LIN {X 0,Y 312.463,Z 248.062,A -85,B 0,C 180,E1 -15613.962,E2 -15613.962} C_VEL
LIN {X 0,Y 312.46,Z 248.062,A -85,B 0,C 180,E1 -15617.921,E2 -15617.921} C_VEL
LIN {X 0,Y 312.479,Z 248.055,A -85,B 0,C 180,E1 -15621.921,E2 -15621.921} C_VEL
LIN {X 0,Y 312.532,Z 248.051,A -85,B 0,C 180,E1 -15624.216,E2 -15624.216} C_VEL
LIN {X 0,Y 312.504,Z 248.056,A -85,B 0,C 180,E1 -15627.33,E2 -15627.33} C_VEL
LIN {X 0,Y 312.506,Z 248.055,A -85,B 0,C 180,E1 -15631.289,E2 -15631.289} C_VEL
LIN {X 0,Y 312.546,Z 248.054,A -85,B 0,C 180,E1 -15634.704,E2 -15634.704} C_VEL
LIN {X 0,Y 312.532,Z 248.054,A -85,B 0,C 180,E1 -15638.908,E2 -15638.908} C_VEL
LIN {X 0,Y 312.587,Z 248.036,A -85,B 0,C 180,E1 -15641.649,E2 -15641.649} C_VEL
LIN {X 0,Y 312.682,Z 248.028,A -85,B 0,C 180,E1 -15645.682,E2 -15645.682} C_VEL
LIN {X 0,Y 312.68,Z 248.034,A -85,B 0,C 180,E1 -15649.637,E2 -15649.637} C_VEL
LIN {X 0,Y 312.811,Z 248.012,A -85,B 0,C 180,E1 -15652.249,E2 -15652.249} C_VEL
LIN {X 0,Y 312.682,Z 248.035,A -85,B 0,C 180,E1 -15654.838,E2 -15654.838} C_VEL
LIN {X 0,Y 312.97,Z 247.999,A -85,B 0,C 180,E1 -15658.709,E2 -15658.709} C_VEL
LIN {X 0,Y 312.953,Z 247.992,A -85,B 0,C 180,E1 -15661.282,E2 -15661.282} C_VEL
LIN {X 0,Y 312.826,Z 248.014,A -85,B 0,C 180,E1 -15666.445,E2 -15666.445} C_VEL
LIN {X 0,Y 312.738,Z 248.025,A -85,B 0,C 180,E1 -15669.046,E2 -15669.046} C_VEL
LIN {X 0,Y 312.618,Z 248.04,A -85,B 0,C 180,E1 -15672.987,E2 -15672.987} C_VEL
LIN {X 0,Y 312.61,Z 248.048,A -85,B 0,C 180,E1 -15675.646,E2 -15675.646} C_VEL
LIN {X 0,Y 312.547,Z 248.051,A -85,B 0,C 180,E1 -15679.707,E2 -15679.707} C_VEL
LIN {X 0,Y 312.504,Z 248.054,A -85,B 0,C 180,E1 -15682.775,E2 -15682.775} C_VEL
LIN {X 0,Y 312.511,Z 248.055,A -85,B 0,C 180,E1 -15685.904,E2 -15685.904} C_VEL
LIN {X 0,Y 312.474,Z 248.056,A -85,B 0,C 180,E1 -15689.651,E2 -15689.651} C_VEL
LIN {X 0,Y 312.496,Z 248.061,A -85,B 0,C 180,E1 -15693.685,E2 -15693.685} C_VEL
LIN {X 0,Y 312.517,Z 248.195,A -85,B 0,C 180,E1 -15696.503,E2 -15696.503} C_VEL
LIN {X 0,Y 314.901,Z 258.143,A -85,B 0,C 180,E1 -15699.907,E2 -15699.907} C_VEL
LIN {X 0,Y 315.377,Z 260.256,A -85,B 0,C 180,E1 -15700.485,E2 -15700.485} C_VEL
LIN {X 0,Y 322.558,Z 277.103,A -85,B 0,C 180,E1 -15701.66,E2 -15701.66} C_VEL
LIN {X 0,Y 325.828,Z 294.759,A -85,B 0,C 180,E1 -15702.408,E2 -15702.408} C_VEL
LIN {X 0,Y 323.737,Z 367.932,A -85,B 0,C 180,E1 -15704.094,E2 -15704.094} C_VEL
LIN {X 0,Y 322.887,Z 381.785,A -85,B 0,C 180,E1 -15704.674,E2 -15704.674} C_VEL
LIN {X 0,Y 321.877,Z 394.277,A -85,B 0,C 180,E1 -15705.46,E2 -15705.46} C_VEL
LIN {X 0,Y 320.612,Z 405.801,A -85,B 0,C 180,E1 -15706.439,E2 -15706.439} C_VEL
LIN {X 0,Y 319.215,Z 416.53,A -85,B 0,C 180,E1 -15707.605,E2 -15707.605} C_VEL
LIN {X 0,Y 317.574,Z 427.06,A -85,B 0,C 180,E1 -15709.033,E2 -15709.033} C_VEL
LIN {X 0,Y 316.045,Z 436.49,A -85,B 0,C 180,E1 -15710.635,E2 -15710.635} C_VEL
LIN {X 0,Y 314.588,Z 445.259,A -85,B 0,C 180,E1 -15712.501,E2 -15712.501} C_VEL
LIN {X 0,Y 313.392,Z 452.216,A -85,B 0,C 180,E1 -15714.335,E2 -15714.335} C_VEL
LIN {X 0,Y 312.34,Z 458.327,A -85,B 0,C 180,E1 -15716.35,E2 -15716.35} C_VEL
LIN {X 0,Y 311.51,Z 463.814,A -85,B 0,C 180,E1 -15718.743,E2 -15718.743} C_VEL
LIN {X 0,Y 311.136,Z 466.376,A -85,B 0,C 180,E1 -15720.204,E2 -15720.204} C_VEL
LIN {X 0,Y 310.784,Z 468.579,A -85,B 0,C 180,E1 -15721.864,E2 -15721.864} C_VEL
LIN {X 0,Y 310.578,Z 469.776,A -85,B 0,C 180,E1 -15723.092,E2 -15723.092} C_VEL
LIN {X 0,Y 310.4,Z 470.87,A -85,B 0,C 180,E1 -15724.899,E2 -15724.899} C_VEL
LIN {X 0,Y 310.274,Z 471.125,A -85,B 0,C 180,E1 -15727.354,E2 -15727.354} C_VEL
LIN {X 0,Y 310.36,Z 470.641,A -85,B 0,C 180,E1 -15728.759,E2 -15728.759} C_VEL
LIN {X 0,Y 310.458,Z 469.66,A -85,B 0,C 180,E1 -15730.151,E2 -15730.151} C_VEL
LIN {X 0,Y 310.677,Z 467.93,A -85,B 0,C 180,E1 -15731.804,E2 -15731.804} C_VEL
LIN {X 0,Y 310.973,Z 465.238,A -85,B 0,C 180,E1 -15733.592,E2 -15733.592} C_VEL
LIN {X 0,Y 311.569,Z 460.486,A -85,B 0,C 180,E1 -15735.89,E2 -15735.89} C_VEL
LIN {X 0,Y 312.285,Z 454.707,A -85,B 0,C 180,E1 -15737.986,E2 -15737.986} C_VEL
LIN {X 0,Y 313.308,Z 447.063,A -85,B 0,C 180,E1 -15740.153,E2 -15740.153} C_VEL
LIN {X 0,Y 314.507,Z 438.905,A -85,B 0,C 180,E1 -15741.973,E2 -15741.973} C_VEL
LIN {X 0,Y 315.903,Z 428.823,A -85,B 0,C 180,E1 -15743.775,E2 -15743.775} C_VEL
LIN {X 0,Y 317.304,Z 418.3,A -85,B 0,C 180,E1 -15745.273,E2 -15745.273} C_VEL
LIN {X 0,Y 318.603,Z 407.173,A -85,B 0,C 180,E1 -15746.523,E2 -15746.523} C_VEL
LIN {X 0,Y 319.848,Z 394.355,A -85,B 0,C 180,E1 -15747.64,E2 -15747.64} C_VEL
LIN {X 0,Y 320.764,Z 381.876,A -85,B 0,C 180,E1 -15748.432,E2 -15748.432} C_VEL
LIN {X 0,Y 321.492,Z 369.025,A -85,B 0,C 180,E1 -15748.983,E2 -15748.983} C_VEL
LIN {X 0,Y 322.286,Z 339.702,A -85,B 0,C 180,E1 -15749.689,E2 -15749.689} C_VEL
LIN {X 0,Y 323.282,Z 292.285,A -85,B 0,C 180,E1 -15750.766,E2 -15750.766} C_VEL
LIN {X 0,Y 319.172,Z 270.918,A -85,B 0,C 180,E1 -15751.59,E2 -15751.59} C_VEL
LIN {X 0,Y 315.333,Z 260.355,A -85,B 0,C 180,E1 -15752.181,E2 -15752.181} C_VEL
LIN {X 0,Y 314.589,Z 256.888,A -85,B 0,C 180,E1 -15753.203,E2 -15753.203} C_VEL
LIN {X 0,Y 312.881,Z 248.091,A -85,B 0,C 180,E1 -15756.207,E2 -15756.207} C_VEL
LIN {X 0,Y 312.734,Z 248.024,A -85,B 0,C 180,E1 -15759.052,E2 -15759.052} C_VEL
LIN {X 0,Y 312.603,Z 248.034,A -85,B 0,C 180,E1 -15762.993,E2 -15762.993} C_VEL
LIN {X 0,Y 312.607,Z 248.043,A -85,B 0,C 180,E1 -15765.652,E2 -15765.652} C_VEL
LIN {X 0,Y 312.578,Z 248.046,A -85,B 0,C 180,E1 -15769.227,E2 -15769.227} C_VEL
LIN {X 0,Y 312.492,Z 248.057,A -85,B 0,C 180,E1 -15772.781,E2 -15772.781} C_VEL
LIN {X 0,Y 312.502,Z 248.057,A -85,B 0,C 180,E1 -15775.911,E2 -15775.911} C_VEL
LIN {X 0,Y 312.445,Z 248.051,A -85,B 0,C 180,E1 -15779.661,E2 -15779.661} C_VEL
LIN {X 0,Y 312.494,Z 248.056,A -85,B 0,C 180,E1 -15783.693,E2 -15783.693} C_VEL
LIN {X 0,Y 312.485,Z 248.057,A -85,B 0,C 180,E1 -15787.392,E2 -15787.392} C_VEL
LIN {X 0,Y 312.402,Z 248.056,A -85,B 0,C 180,E1 -15791.155,E2 -15791.155} C_VEL
LIN {X 0,Y 311.733,Z 248.136,A -85,B 0,C 180,E1 -15792.231,E2 -15792.231} C_VEL
LIN {X 0,Y 308.889,Z 248.495,A -85,B 0,C 180,E1 -15793.983,E2 -15793.983} C_VEL
LIN {X 0,Y 306.488,Z 248.805,A -85,B 0,C 180,E1 -15795.404,E2 -15795.404} C_VEL
LIN {X 0,Y 305.47,Z 248.934,A -85,B 0,C 180,E1 -15796.504,E2 -15796.504} C_VEL
LIN {X 0,Y 305.394,Z 248.94,A -85,B 0,C 180,E1 -15796.877,E2 -15796.877} C_VEL
LIN {X 0,Y 305.392,Z 248.928,A -85,B 0,C 180,E1 -15799.889,E2 -15799.889} C_VEL
LIN {X 0,Y 305.446,Z 248.929,A -85,B 0,C 180,E1 -15803.642,E2 -15803.642} C_VEL
LIN {X 0,Y 305.451,Z 248.935,A -85,B 0,C 180,E1 -15806.488,E2 -15806.488} C_VEL
LIN {X 0,Y 305.404,Z 248.92,A -85,B 0,C 180,E1 -15809.591,E2 -15809.591} C_VEL
LIN {X 0,Y 305.43,Z 248.914,A -85,B 0,C 180,E1 -15812.606,E2 -15812.606} C_VEL
LIN {X 0,Y 305.446,Z 248.936,A -85,B 0,C 180,E1 -15815.539,E2 -15815.539} C_VEL
LIN {X 0,Y 305.489,Z 248.916,A -85,B 0,C 180,E1 -15819.818,E2 -15819.818} C_VEL
LIN {X 0,Y 305.536,Z 248.886,A -85,B 0,C 180,E1 -15822.606,E2 -15822.606} C_VEL
LIN {X 0,Y 305.622,Z 248.9,A -85,B 0,C 180,E1 -15825.353,E2 -15825.353} C_VEL
LIN {X 0,Y 305.621,Z 248.914,A -85,B 0,C 180,E1 -15829.404,E2 -15829.404} C_VEL
LIN {X 0,Y 305.745,Z 248.876,A -85,B 0,C 180,E1 -15832.077,E2 -15832.077} C_VEL
LIN {X 0,Y 305.657,Z 248.877,A -85,B 0,C 180,E1 -15834.728,E2 -15834.728} C_VEL
LIN {X 0,Y 305.937,Z 248.873,A -85,B 0,C 180,E1 -15838.688,E2 -15838.688} C_VEL
LIN {X 0,Y 305.947,Z 248.868,A -85,B 0,C 180,E1 -15841.321,E2 -15841.321} C_VEL
LIN {X 0,Y 305.809,Z 248.866,A -85,B 0,C 180,E1 -15846.603,E2 -15846.603} C_VEL
LIN {X 0,Y 305.701,Z 248.902,A -85,B 0,C 180,E1 -15849.265,E2 -15849.265} C_VEL
LIN {X 0,Y 305.593,Z 248.905,A -85,B 0,C 180,E1 -15853.3,E2 -15853.3} C_VEL
LIN {X 0,Y 305.56,Z 248.898,A -85,B 0,C 180,E1 -15856.026,E2 -15856.026} C_VEL
LIN {X 0,Y 305.552,Z 248.923,A -85,B 0,C 180,E1 -15859.43,E2 -15859.43} C_VEL
LIN {X 0,Y 305.497,Z 248.911,A -85,B 0,C 180,E1 -15863.042,E2 -15863.042} C_VEL
LIN {X 0,Y 305.481,Z 248.926,A -85,B 0,C 180,E1 -15866.2,E2 -15866.2} C_VEL
LIN {X 0,Y 305.46,Z 248.933,A -85,B 0,C 180,E1 -15869.036,E2 -15869.036} C_VEL
LIN {X 0,Y 305.448,Z 248.924,A -85,B 0,C 180,E1 -15871.956,E2 -15871.956} C_VEL
LIN {X 0,Y 305.474,Z 248.936,A -85,B 0,C 180,E1 -15875.116,E2 -15875.116} C_VEL
LIN {X 0,Y 305.446,Z 248.93,A -85,B 0,C 180,E1 -15878.527,E2 -15878.527} C_VEL
LIN {X 0,Y 305.448,Z 248.925,A -85,B 0,C 180,E1 -15882.583,E2 -15882.583} C_VEL
LIN {X 0,Y 305.434,Z 248.933,A -85,B 0,C 180,E1 -15886.345,E2 -15886.345} C_VEL
LIN {X 0,Y 305.424,Z 248.938,A -85,B 0,C 180,E1 -15889.886,E2 -15889.886} C_VEL
LIN {X 0,Y 305.476,Z 248.933,A -85,B 0,C 180,E1 -15893.638,E2 -15893.638} C_VEL
LIN {X 0,Y 305.479,Z 248.924,A -85,B 0,C 180,E1 -15896.484,E2 -15896.484} C_VEL
LIN {X 0,Y 305.471,Z 248.993,A -85,B 0,C 180,E1 -15898.211,E2 -15898.211} C_VEL
LIN {X 0,Y 307.479,Z 258.119,A -85,B 0,C 180,E1 -15901.314,E2 -15901.314} C_VEL
LIN {X 0,Y 309.395,Z 267.921,A -85,B 0,C 180,E1 -15904.363,E2 -15904.363} C_VEL
LIN {X 0,Y 310.742,Z 272.023,A -85,B 0,C 180,E1 -15904.643,E2 -15904.643} C_VEL
LIN {X 0,Y 315.958,Z 302.066,A -85,B 0,C 180,E1 -15905.787,E2 -15905.787} C_VEL
LIN {X 0,Y 316.558,Z 306.759,A -85,B 0,C 180,E1 -15905.946,E2 -15905.946} C_VEL
LIN {X 0,Y 314.819,Z 376.369,A -85,B 0,C 180,E1 -15907.581,E2 -15907.581} C_VEL
LIN {X 0,Y 314.013,Z 389.829,A -85,B 0,C 180,E1 -15908.155,E2 -15908.155} C_VEL
LIN {X 0,Y 312.93,Z 402.282,A -85,B 0,C 180,E1 -15908.939,E2 -15908.939} C_VEL
LIN {X 0,Y 311.745,Z 413.411,A -85,B 0,C 180,E1 -15909.891,E2 -15909.891} C_VEL
LIN {X 0,Y 310.33,Z 425.013,A -85,B 0,C 180,E1 -15911.172,E2 -15911.172} C_VEL
LIN {X 0,Y 308.952,Z 435.464,A -85,B 0,C 180,E1 -15912.628,E2 -15912.628} C_VEL
LIN {X 0,Y 307.797,Z 444.002,A -85,B 0,C 180,E1 -15914.097,E2 -15914.097} C_VEL
LIN {X 0,Y 306.403,Z 453.236,A -85,B 0,C 180,E1 -15916.063,E2 -15916.063} C_VEL
LIN {X 0,Y 305.282,Z 460.656,A -85,B 0,C 180,E1 -15918.041,E2 -15918.041} C_VEL
LIN {X 0,Y 304.54,Z 466.605,A -85,B 0,C 180,E1 -15920.032,E2 -15920.032} C_VEL
LIN {X 0,Y 304.022,Z 471.29,A -85,B 0,C 180,E1 -15922.026,E2 -15922.026} C_VEL
LIN {X 0,Y 303.673,Z 475.387,A -85,B 0,C 180,E1 -15924.387,E2 -15924.387} C_VEL
LIN {X 0,Y 303.596,Z 477.39,A -85,B 0,C 180,E1 -15926.017,E2 -15926.017} C_VEL
LIN {X 0,Y 303.586,Z 478.574,A -85,B 0,C 180,E1 -15927.345,E2 -15927.345} C_VEL
LIN {X 0,Y 303.534,Z 479.309,A -85,B 0,C 180,E1 -15928.672,E2 -15928.672} C_VEL
LIN {X 0,Y 303.541,Z 479.653,A -85,B 0,C 180,E1 -15929.999,E2 -15929.999} C_VEL
LIN {X 0,Y 303.534,Z 479.61,A -85,B 0,C 180,E1 -15931.326,E2 -15931.326} C_VEL
LIN {X 0,Y 303.588,Z 479.175,A -85,B 0,C 180,E1 -15932.653,E2 -15932.653} C_VEL
LIN {X 0,Y 303.606,Z 478.302,A -85,B 0,C 180,E1 -15933.981,E2 -15933.981} C_VEL
LIN {X 0,Y 303.849,Z 475.356,A -85,B 0,C 180,E1 -15936.64,E2 -15936.64} C_VEL
LIN {X 0,Y 304.242,Z 471.997,A -85,B 0,C 180,E1 -15938.634,E2 -15938.634} C_VEL
LIN {X 0,Y 304.898,Z 467.57,A -85,B 0,C 180,E1 -15940.625,E2 -15940.625} C_VEL
LIN {X 0,Y 305.793,Z 461.955,A -85,B 0,C 180,E1 -15942.61,E2 -15942.61} C_VEL
LIN {X 0,Y 307.091,Z 454.946,A -85,B 0,C 180,E1 -15944.579,E2 -15944.579} C_VEL
LIN {X 0,Y 308.657,Z 446.316,A -85,B 0,C 180,E1 -15946.507,E2 -15946.507} C_VEL
LIN {X 0,Y 310.224,Z 436.252,A -85,B 0,C 180,E1 -15948.319,E2 -15948.319} C_VEL
LIN {X 0,Y 311.905,Z 426.151,A -85,B 0,C 180,E1 -15949.753,E2 -15949.753} C_VEL
LIN {X 0,Y 313.56,Z 414.959,A -85,B 0,C 180,E1 -15951.014,E2 -15951.014} C_VEL
LIN {X 0,Y 315.056,Z 402.422,A -85,B 0,C 180,E1 -15952.112,E2 -15952.112} C_VEL
LIN {X 0,Y 316.337,Z 389.519,A -85,B 0,C 180,E1 -15952.921,E2 -15952.921} C_VEL
LIN {X 0,Y 317.264,Z 375.829,A -85,B 0,C 180,E1 -15953.498,E2 -15953.498} C_VEL
LIN {X 0,Y 319.018,Z 315.952,A -85,B 0,C 180,E1 -15954.913,E2 -15954.913} C_VEL
LIN {X 0,Y 319.112,Z 306.429,A -85,B 0,C 180,E1 -15955.15,E2 -15955.15} C_VEL
LIN {X 0,Y 315.545,Z 285.854,A -85,B 0,C 180,E1 -15956.032,E2 -15956.032} C_VEL
LIN {X 0,Y 313.593,Z 277.044,A -85,B 0,C 180,E1 -15956.463,E2 -15956.463} C_VEL
LIN {X 0,Y 309.713,Z 267.394,A -85,B 0,C 180,E1 -15957.172,E2 -15957.172} C_VEL
LIN {X 0,Y 307.708,Z 258.136,A -85,B 0,C 180,E1 -15960.162,E2 -15960.162} C_VEL
LIN {X 0,Y 305.518,Z 248.992,A -85,B 0,C 180,E1 -15963.459,E2 -15963.459} C_VEL
LIN {X 0,Y 305.461,Z 248.927,A -85,B 0,C 180,E1 -15966.74,E2 -15966.74} C_VEL
LIN {X 0,Y 305.416,Z 248.93,A -85,B 0,C 180,E1 -15970.587,E2 -15970.587} C_VEL
LIN {X 0,Y 305.427,Z 248.936,A -85,B 0,C 180,E1 -15973.653,E2 -15973.653} C_VEL
LIN {X 0,Y 305.44,Z 248.938,A -85,B 0,C 180,E1 -15977.415,E2 -15977.415} C_VEL
LIN {X 0,Y 305.445,Z 248.93,A -85,B 0,C 180,E1 -15981.589,E2 -15981.589} C_VEL
LIN {X 0,Y 305.464,Z 248.929,A -85,B 0,C 180,E1 -15984.883,E2 -15984.883} C_VEL
LIN {X 0,Y 305.444,Z 248.931,A -85,B 0,C 180,E1 -15988.355,E2 -15988.355} C_VEL
LIN {X 0,Y 305.475,Z 248.932,A -85,B 0,C 180,E1 -15991.105,E2 -15991.105} C_VEL
LIN {X 0,Y 305.498,Z 248.927,A -85,B 0,C 180,E1 -15994.077,E2 -15994.077} C_VEL
LIN {X 0,Y 305.474,Z 248.924,A -85,B 0,C 180,E1 -15996.972,E2 -15996.972} C_VEL
LIN {X 0,Y 305.547,Z 248.914,A -85,B 0,C 180,E1 -16001.211,E2 -16001.211} C_VEL
LIN {X 0,Y 305.623,Z 248.909,A -85,B 0,C 180,E1 -16005.344,E2 -16005.344} C_VEL
LIN {X 0,Y 305.619,Z 248.916,A -85,B 0,C 180,E1 -16009.395,E2 -16009.395} C_VEL
LIN {X 0,Y 305.757,Z 248.889,A -85,B 0,C 180,E1 -16012.069,E2 -16012.069} C_VEL
LIN {X 0,Y 305.653,Z 248.911,A -85,B 0,C 180,E1 -16014.719,E2 -16014.719} C_VEL
LIN {X 0,Y 305.936,Z 248.875,A -85,B 0,C 180,E1 -16018.679,E2 -16018.679} C_VEL
LIN {X 0,Y 305.921,Z 248.868,A -85,B 0,C 180,E1 -16021.312,E2 -16021.312} C_VEL
LIN {X 0,Y 305.771,Z 248.894,A -85,B 0,C 180,E1 -16026.594,E2 -16026.594} C_VEL
LIN {X 0,Y 305.681,Z 248.902,A -85,B 0,C 180,E1 -16029.257,E2 -16029.257} C_VEL
LIN {X 0,Y 305.57,Z 248.917,A -85,B 0,C 180,E1 -16033.292,E2 -16033.292} C_VEL
LIN {X 0,Y 305.539,Z 248.925,A -85,B 0,C 180,E1 -16036.018,E2 -16036.018} C_VEL
LIN {X 0,Y 305.53,Z 248.927,A -85,B 0,C 180,E1 -16039.424,E2 -16039.424} C_VEL
LIN {X 0,Y 305.468,Z 248.93,A -85,B 0,C 180,E1 -16043.035,E2 -16043.035} C_VEL
LIN {X 0,Y 305.451,Z 248.937,A -85,B 0,C 180,E1 -16046.193,E2 -16046.193} C_VEL
LIN {X 0,Y 305.427,Z 248.928,A -85,B 0,C 180,E1 -16049.03,E2 -16049.03} C_VEL
LIN {X 0,Y 305.414,Z 248.933,A -85,B 0,C 180,E1 -16051.949,E2 -16051.949} C_VEL
LIN {X 0,Y 305.515,Z 249.124,A -85,B 0,C 180,E1 -16055.913,E2 -16055.913} C_VEL
LIN {X 0,Y 307.844,Z 258.921,A -85,B 0,C 180,E1 -16059.366,E2 -16059.366} C_VEL
LIN {X 0,Y 308.209,Z 260.311,A -85,B 0,C 180,E1 -16059.734,E2 -16059.734} C_VEL
LIN {X 0,Y 315.471,Z 276.995,A -85,B 0,C 180,E1 -16060.969,E2 -16060.969} C_VEL
LIN {X 0,Y 316.962,Z 281.432,A -85,B 0,C 180,E1 -16061.233,E2 -16061.233} C_VEL
LIN {X 0,Y 319.506,Z 295.751,A -85,B 0,C 180,E1 -16061.852,E2 -16061.852} C_VEL
LIN {X 0,Y 317.415,Z 367.051,A -85,B 0,C 180,E1 -16063.522,E2 -16063.522} C_VEL
LIN {X 0,Y 316.594,Z 380.179,A -85,B 0,C 180,E1 -16064.056,E2 -16064.056} C_VEL
LIN {X 0,Y 315.55,Z 392.768,A -85,B 0,C 180,E1 -16064.828,E2 -16064.828} C_VEL
LIN {X 0,Y 314.231,Z 404.522,A -85,B 0,C 180,E1 -16065.801,E2 -16065.801} C_VEL
LIN {X 0,Y 312.784,Z 415.314,A -85,B 0,C 180,E1 -16066.963,E2 -16066.963} C_VEL
LIN {X 0,Y 311.074,Z 426.08,A -85,B 0,C 180,E1 -16068.419,E2 -16068.419} C_VEL
LIN {X 0,Y 309.412,Z 435.917,A -85,B 0,C 180,E1 -16070.085,E2 -16070.085} C_VEL
LIN {X 0,Y 307.858,Z 444.664,A -85,B 0,C 180,E1 -16071.95,E2 -16071.95} C_VEL
LIN {X 0,Y 306.598,Z 451.752,A -85,B 0,C 180,E1 -16073.827,E2 -16073.827} C_VEL
LIN {X 0,Y 305.474,Z 458.032,A -85,B 0,C 180,E1 -16075.908,E2 -16075.908} C_VEL
LIN {X 0,Y 304.649,Z 462.849,A -85,B 0,C 180,E1 -16077.956,E2 -16077.956} C_VEL
LIN {X 0,Y 304.038,Z 466.792,A -85,B 0,C 180,E1 -16080.201,E2 -16080.201} C_VEL
LIN {X 0,Y 303.579,Z 469.427,A -85,B 0,C 180,E1 -16082.42,E2 -16082.42} C_VEL
LIN {X 0,Y 303.329,Z 470.904,A -85,B 0,C 180,E1 -16084.622,E2 -16084.622} C_VEL
LIN {X 0,Y 303.181,Z 471.291,A -85,B 0,C 180,E1 -16086.793,E2 -16086.793} C_VEL
LIN {X 0,Y 303.252,Z 470.953,A -85,B 0,C 180,E1 -16088.236,E2 -16088.236} C_VEL
LIN {X 0,Y 303.305,Z 470.184,A -85,B 0,C 180,E1 -16089.663,E2 -16089.663} C_VEL
LIN {X 0,Y 303.564,Z 468.295,A -85,B 0,C 180,E1 -16091.641,E2 -16091.641} C_VEL
LIN {X 0,Y 303.933,Z 465.019,A -85,B 0,C 180,E1 -16093.891,E2 -16093.891} C_VEL
LIN {X 0,Y 304.581,Z 460.129,A -85,B 0,C 180,E1 -16096.237,E2 -16096.237} C_VEL
LIN {X 0,Y 305.339,Z 454.229,A -85,B 0,C 180,E1 -16098.382,E2 -16098.382} C_VEL
LIN {X 0,Y 306.383,Z 446.861,A -85,B 0,C 180,E1 -16100.487,E2 -16100.487} C_VEL
LIN {X 0,Y 307.698,Z 438.079,A -85,B 0,C 180,E1 -16102.455,E2 -16102.455} C_VEL
LIN {X 0,Y 309.063,Z 428.803,A -85,B 0,C 180,E1 -16104.128,E2 -16104.128} C_VEL
LIN {X 0,Y 310.411,Z 418.956,A -85,B 0,C 180,E1 -16105.566,E2 -16105.566} C_VEL
LIN {X 0,Y 311.855,Z 407.074,A -85,B 0,C 180,E1 -16106.933,E2 -16106.933} C_VEL
LIN {X 0,Y 313.045,Z 395.22,A -85,B 0,C 180,E1 -16107.991,E2 -16107.991} C_VEL
LIN {X 0,Y 313.998,Z 383.123,A -85,B 0,C 180,E1 -16108.799,E2 -16108.799} C_VEL
LIN {X 0,Y 314.79,Z 369.706,A -85,B 0,C 180,E1 -16109.401,E2 -16109.401} C_VEL
LIN {X 0,Y 315.518,Z 347.471,A -85,B 0,C 180,E1 -16109.961,E2 -16109.961} C_VEL
LIN {X 0,Y 316.669,Z 293.156,A -85,B 0,C 180,E1 -16111.224,E2 -16111.224} C_VEL
LIN {X 0,Y 312.829,Z 273.23,A -85,B 0,C 180,E1 -16112.013,E2 -16112.013} C_VEL
LIN {X 0,Y 308.164,Z 260.505,A -85,B 0,C 180,E1 -16112.738,E2 -16112.738} C_VEL
LIN {X 0,Y 307.685,Z 258.533,A -85,B 0,C 180,E1 -16113.275,E2 -16113.275} C_VEL
LIN {X 0,Y 305.844,Z 248.989,A -85,B 0,C 180,E1 -16116.599,E2 -16116.599} C_VEL
LIN {X 0,Y 305.671,Z 248.903,A -85,B 0,C 180,E1 -16119.263,E2 -16119.263} C_VEL
LIN {X 0,Y 305.557,Z 248.913,A -85,B 0,C 180,E1 -16123.298,E2 -16123.298} C_VEL
LIN {X 0,Y 305.562,Z 248.918,A -85,B 0,C 180,E1 -16126.023,E2 -16126.023} C_VEL
LIN {X 0,Y 305.529,Z 248.922,A -85,B 0,C 180,E1 -16129.438,E2 -16129.438} C_VEL
LIN {X 0,Y 305.457,Z 248.933,A -85,B 0,C 180,E1 -16133.043,E2 -16133.043} C_VEL
LIN {X 0,Y 305.442,Z 248.939,A -85,B 0,C 180,E1 -16136.201,E2 -16136.201} C_VEL
LIN {X 0,Y 305.408,Z 248.927,A -85,B 0,C 180,E1 -16139.033,E2 -16139.033} C_VEL
LIN {X 0,Y 305.409,Z 248.942,A -85,B 0,C 180,E1 -16141.957,E2 -16141.957} C_VEL
LIN {X 0,Y 305.435,Z 248.92,A -85,B 0,C 180,E1 -16145.118,E2 -16145.118} C_VEL
LIN {X 0,Y 305.41,Z 248.944,A -85,B 0,C 180,E1 -16148.529,E2 -16148.529} C_VEL
LIN {X 0,Y 305.412,Z 248.921,A -85,B 0,C 180,E1 -16152.586,E2 -16152.586} C_VEL
LIN {X 0,Y 305.394,Z 248.94,A -85,B 0,C 180,E1 -16156.877,E2 -16156.877} C_VEL
LIN {X 0,Y 304.737,Z 249.024,A -85,B 0,C 180,E1 -16157.978,E2 -16157.978} C_VEL
LIN {X 0,Y 301.874,Z 249.366,A -85,B 0,C 180,E1 -16159.771,E2 -16159.771} C_VEL
LIN {X 0,Y 299.457,Z 249.659,A -85,B 0,C 180,E1 -16161.226,E2 -16161.226} C_VEL
LIN {X 0,Y 298.447,Z 249.785,A -85,B 0,C 180,E1 -16162.353,E2 -16162.353} C_VEL
LIN {X 0,Y 298.38,Z 249.796,A -85,B 0,C 180,E1 -16162.735,E2 -16162.735} C_VEL
LIN {X 0,Y 298.393,Z 249.814,A -85,B 0,C 180,E1 -16165.586,E2 -16165.586} C_VEL
LIN {X 0,Y 298.359,Z 249.807,A -85,B 0,C 180,E1 -16168.794,E2 -16168.794} C_VEL
LIN {X 0,Y 298.384,Z 249.785,A -85,B 0,C 180,E1 -16171.902,E2 -16171.902} C_VEL
LIN {X 0,Y 298.412,Z 249.806,A -85,B 0,C 180,E1 -16174.923,E2 -16174.923} C_VEL
LIN {X 0,Y 298.419,Z 249.801,A -85,B 0,C 180,E1 -16179.319,E2 -16179.319} C_VEL
LIN {X 0,Y 298.472,Z 249.766,A -85,B 0,C 180,E1 -16182.181,E2 -16182.181} C_VEL
LIN {X 0,Y 298.583,Z 249.775,A -85,B 0,C 180,E1 -16184.999,E2 -16184.999} C_VEL
LIN {X 0,Y 298.58,Z 249.79,A -85,B 0,C 180,E1 -16189.151,E2 -16189.151} C_VEL
LIN {X 0,Y 298.696,Z 249.755,A -85,B 0,C 180,E1 -16191.889,E2 -16191.889} C_VEL
LIN {X 0,Y 298.627,Z 249.751,A -85,B 0,C 180,E1 -16194.603,E2 -16194.603} C_VEL
LIN {X 0,Y 298.905,Z 249.749,A -85,B 0,C 180,E1 -16198.657,E2 -16198.657} C_VEL
LIN {X 0,Y 298.914,Z 249.745,A -85,B 0,C 180,E1 -16201.352,E2 -16201.352} C_VEL
LIN {X 0,Y 298.758,Z 249.746,A -85,B 0,C 180,E1 -16206.759,E2 -16206.759} C_VEL
LIN {X 0,Y 298.632,Z 249.783,A -85,B 0,C 180,E1 -16209.486,E2 -16209.486} C_VEL
LIN {X 0,Y 298.552,Z 249.781,A -85,B 0,C 180,E1 -16213.62,E2 -16213.62} C_VEL
LIN {X 0,Y 298.495,Z 249.78,A -85,B 0,C 180,E1 -16216.416,E2 -16216.416} C_VEL
LIN {X 0,Y 298.493,Z 249.802,A -85,B 0,C 180,E1 -16219.642,E2 -16219.642} C_VEL
LIN {X 0,Y 298.431,Z 249.786,A -85,B 0,C 180,E1 -16223.604,E2 -16223.604} C_VEL
LIN {X 0,Y 298.419,Z 249.807,A -85,B 0,C 180,E1 -16226.585,E2 -16226.585} C_VEL
LIN {X 0,Y 298.405,Z 249.806,A -85,B 0,C 180,E1 -16229.647,E2 -16229.647} C_VEL
LIN {X 0,Y 298.405,Z 249.805,A -85,B 0,C 180,E1 -16232.803,E2 -16232.803} C_VEL
LIN {X 0,Y 298.439,Z 249.801,A -85,B 0,C 180,E1 -16236.804,E2 -16236.804} C_VEL
LIN {X 0,Y 298.387,Z 249.816,A -85,B 0,C 180,E1 -16239.494,E2 -16239.494} C_VEL
LIN {X 0,Y 298.383,Z 249.807,A -85,B 0,C 180,E1 -16243.099,E2 -16243.099} C_VEL
LIN {X 0,Y 298.384,Z 249.812,A -85,B 0,C 180,E1 -16246.916,E2 -16246.916} C_VEL
LIN {X 0,Y 298.399,Z 249.816,A -85,B 0,C 180,E1 -16251.012,E2 -16251.012} C_VEL
LIN {X 0,Y 298.418,Z 249.812,A -85,B 0,C 180,E1 -16253.929,E2 -16253.929} C_VEL
LIN {X 0,Y 298.417,Z 249.875,A -85,B 0,C 180,E1 -16257.768,E2 -16257.768} C_VEL
LIN {X 0,Y 300.444,Z 259.031,A -85,B 0,C 180,E1 -16260.961,E2 -16260.961} C_VEL
LIN {X 0,Y 302.159,Z 267.831,A -85,B 0,C 180,E1 -16263.772,E2 -16263.772} C_VEL
LIN {X 0,Y 303.904,Z 272.76,A -85,B 0,C 180,E1 -16264.112,E2 -16264.112} C_VEL
LIN {X 0,Y 305.261,Z 278.652,A -85,B 0,C 180,E1 -16264.375,E2 -16264.375} C_VEL
LIN {X 0,Y 309.848,Z 306.247,A -85,B 0,C 180,E1 -16265.437,E2 -16265.437} C_VEL
LIN {X 0,Y 308.263,Z 373.719,A -85,B 0,C 180,E1 -16267.048,E2 -16267.048} C_VEL
LIN {X 0,Y 307.527,Z 387.205,A -85,B 0,C 180,E1 -16267.581,E2 -16267.581} C_VEL
LIN {X 0,Y 306.39,Z 400.316,A -85,B 0,C 180,E1 -16268.379,E2 -16268.379} C_VEL
LIN {X 0,Y 305.051,Z 412.78,A -85,B 0,C 180,E1 -16269.43,E2 -16269.43} C_VEL
LIN {X 0,Y 303.574,Z 424.482,A -85,B 0,C 180,E1 -16270.736,E2 -16270.736} C_VEL
LIN {X 0,Y 302.152,Z 435.01,A -85,B 0,C 180,E1 -16272.224,E2 -16272.224} C_VEL
LIN {X 0,Y 300.937,Z 443.612,A -85,B 0,C 180,E1 -16273.724,E2 -16273.724} C_VEL
LIN {X 0,Y 299.729,Z 451.536,A -85,B 0,C 180,E1 -16275.399,E2 -16275.399} C_VEL
LIN {X 0,Y 298.499,Z 459.256,A -85,B 0,C 180,E1 -16277.42,E2 -16277.42} C_VEL
LIN {X 0,Y 297.514,Z 466.366,A -85,B 0,C 180,E1 -16279.794,E2 -16279.794} C_VEL
LIN {X 0,Y 296.973,Z 471.083,A -85,B 0,C 180,E1 -16281.836,E2 -16281.836} C_VEL
LIN {X 0,Y 296.749,Z 473.599,A -85,B 0,C 180,E1 -16283.198,E2 -16283.198} C_VEL
LIN {X 0,Y 296.565,Z 475.627,A -85,B 0,C 180,E1 -16284.56,E2 -16284.56} C_VEL
LIN {X 0,Y 296.499,Z 477.238,A -85,B 0,C 180,E1 -16285.921,E2 -16285.921} C_VEL
LIN {X 0,Y 296.491,Z 478.439,A -85,B 0,C 180,E1 -16287.282,E2 -16287.282} C_VEL
LIN {X 0,Y 296.456,Z 479.193,A -85,B 0,C 180,E1 -16288.64,E2 -16288.64} C_VEL
LIN {X 0,Y 296.459,Z 479.549,A -85,B 0,C 180,E1 -16289.999,E2 -16289.999} C_VEL
LIN {X 0,Y 296.456,Z 479.517,A -85,B 0,C 180,E1 -16291.357,E2 -16291.357} C_VEL
LIN {X 0,Y 296.493,Z 479.098,A -85,B 0,C 180,E1 -16292.716,E2 -16292.716} C_VEL
LIN {X 0,Y 296.51,Z 478.246,A -85,B 0,C 180,E1 -16294.076,E2 -16294.076} C_VEL
LIN {X 0,Y 296.599,Z 476.824,A -85,B 0,C 180,E1 -16295.588,E2 -16295.588} C_VEL
LIN {X 0,Y 297.032,Z 473.24,A -85,B 0,C 180,E1 -16298.16,E2 -16298.16} C_VEL
LIN {X 0,Y 297.624,Z 469.208,A -85,B 0,C 180,E1 -16300.2,E2 -16300.2} C_VEL
LIN {X 0,Y 298.696,Z 463.019,A -85,B 0,C 180,E1 -16302.569,E2 -16302.569} C_VEL
LIN {X 0,Y 299.992,Z 456.285,A -85,B 0,C 180,E1 -16304.585,E2 -16304.585} C_VEL
LIN {X 0,Y 301.604,Z 448.112,A -85,B 0,C 180,E1 -16306.545,E2 -16306.545} C_VEL
LIN {X 0,Y 303.046,Z 439.368,A -85,B 0,C 180,E1 -16308.243,E2 -16308.243} C_VEL
LIN {X 0,Y 304.658,Z 429.987,A -85,B 0,C 180,E1 -16309.716,E2 -16309.716} C_VEL
LIN {X 0,Y 306.556,Z 418.382,A -85,B 0,C 180,E1 -16311.165,E2 -16311.165} C_VEL
LIN {X 0,Y 308.049,Z 406.915,A -85,B 0,C 180,E1 -16312.288,E2 -16312.288} C_VEL
LIN {X 0,Y 309.526,Z 393.778,A -85,B 0,C 180,E1 -16313.234,E2 -16313.234} C_VEL
LIN {X 0,Y 310.641,Z 380.543,A -85,B 0,C 180,E1 -16313.897,E2 -16313.897} C_VEL
LIN {X 0,Y 311.336,Z 366.569,A -85,B 0,C 180,E1 -16314.308,E2 -16314.308} C_VEL
LIN {X 0,Y 312.832,Z 307.519,A -85,B 0,C 180,E1 -16315.725,E2 -16315.725} C_VEL
LIN {X 0,Y 309.162,Z 286.21,A -85,B 0,C 180,E1 -16316.668,E2 -16316.668} C_VEL
LIN {X 0,Y 307.655,Z 279.7,A -85,B 0,C 180,E1 -16317.007,E2 -16317.007} C_VEL
LIN {X 0,Y 302.505,Z 267.291,A -85,B 0,C 180,E1 -16317.957,E2 -16317.957} C_VEL
LIN {X 0,Y 300.527,Z 258.329,A -85,B 0,C 180,E1 -16320.961,E2 -16320.961} C_VEL
LIN {X 0,Y 298.467,Z 249.904,A -85,B 0,C 180,E1 -16324.103,E2 -16324.103} C_VEL
LIN {X 0,Y 298.405,Z 249.811,A -85,B 0,C 180,E1 -16327.758,E2 -16327.758} C_VEL
LIN {X 0,Y 298.354,Z 249.815,A -85,B 0,C 180,E1 -16331.265,E2 -16331.265} C_VEL
LIN {X 0,Y 298.361,Z 249.818,A -85,B 0,C 180,E1 -16335.032,E2 -16335.032} C_VEL
LIN {X 0,Y 298.352,Z 249.818,A -85,B 0,C 180,E1 -16338.918,E2 -16338.918} C_VEL
LIN {X 0,Y 298.39,Z 249.812,A -85,B 0,C 180,E1 -16342.234,E2 -16342.234} C_VEL
LIN {X 0,Y 298.41,Z 249.81,A -85,B 0,C 180,E1 -16345.577,E2 -16345.577} C_VEL
LIN {X 0,Y 298.379,Z 249.81,A -85,B 0,C 180,E1 -16348.785,E2 -16348.785} C_VEL
LIN {X 0,Y 298.412,Z 249.809,A -85,B 0,C 180,E1 -16351.895,E2 -16351.895} C_VEL
LIN {X 0,Y 298.438,Z 249.812,A -85,B 0,C 180,E1 -16354.916,E2 -16354.916} C_VEL
LIN {X 0,Y 298.404,Z 249.807,A -85,B 0,C 180,E1 -16357.858,E2 -16357.858} C_VEL
LIN {X 0,Y 298.507,Z 249.795,A -85,B 0,C 180,E1 -16360.75,E2 -16360.75} C_VEL
LIN {X 0,Y 298.584,Z 249.79,A -85,B 0,C 180,E1 -16364.99,E2 -16364.99} C_VEL
LIN {X 0,Y 298.578,Z 249.794,A -85,B 0,C 180,E1 -16369.142,E2 -16369.142} C_VEL
LIN {X 0,Y 298.706,Z 249.766,A -85,B 0,C 180,E1 -16371.88,E2 -16371.88} C_VEL
LIN {X 0,Y 298.623,Z 249.786,A -85,B 0,C 180,E1 -16374.594,E2 -16374.594} C_VEL
LIN {X 0,Y 298.903,Z 249.751,A -85,B 0,C 180,E1 -16378.648,E2 -16378.648} C_VEL
LIN {X 0,Y 298.889,Z 249.743,A -85,B 0,C 180,E1 -16381.343,E2 -16381.343} C_VEL
LIN {X 0,Y 298.72,Z 249.772,A -85,B 0,C 180,E1 -16386.751,E2 -16386.751} C_VEL
LIN {X 0,Y 298.612,Z 249.782,A -85,B 0,C 180,E1 -16389.478,E2 -16389.478} C_VEL
LIN {X 0,Y 298.53,Z 249.793,A -85,B 0,C 180,E1 -16393.611,E2 -16393.611} C_VEL
LIN {X 0,Y 298.474,Z 249.801,A -85,B 0,C 180,E1 -16396.408,E2 -16396.408} C_VEL
LIN {X 0,Y 298.47,Z 249.805,A -85,B 0,C 180,E1 -16399.637,E2 -16399.637} C_VEL
LIN {X 0,Y 298.404,Z 249.812,A -85,B 0,C 180,E1 -16403.596,E2 -16403.596} C_VEL
LIN {X 0,Y 298.388,Z 249.819,A -85,B 0,C 180,E1 -16406.578,E2 -16406.578} C_VEL
LIN {X 0,Y 298.372,Z 249.811,A -85,B 0,C 180,E1 -16409.64,E2 -16409.64} C_VEL
LIN {X 0,Y 298.37,Z 249.812,A -85,B 0,C 180,E1 -16412.797,E2 -16412.797} C_VEL
LIN {X 0,Y 298.406,Z 249.895,A -85,B 0,C 180,E1 -16415.152,E2 -16415.152} C_VEL
LIN {X 0,Y 300.237,Z 257.215,A -85,B 0,C 180,E1 -16417.906,E2 -16417.906} C_VEL
LIN {X 0,Y 300.985,Z 260.338,A -85,B 0,C 180,E1 -16418.914,E2 -16418.914} C_VEL
LIN {X 0,Y 307.712,Z 275.246,A -85,B 0,C 180,E1 -16420.121,E2 -16420.121} C_VEL
LIN {X 0,Y 310.779,Z 282.908,A -85,B 0,C 180,E1 -16420.653,E2 -16420.653} C_VEL
LIN {X 0,Y 313.23,Z 296.224,A -85,B 0,C 180,E1 -16421.256,E2 -16421.256} C_VEL
LIN {X 0,Y 311.009,Z 367.93,A -85,B 0,C 180,E1 -16422.975,E2 -16422.975} C_VEL
LIN {X 0,Y 310.062,Z 381.697,A -85,B 0,C 180,E1 -16423.565,E2 -16423.565} C_VEL
LIN {X 0,Y 309.004,Z 393.948,A -85,B 0,C 180,E1 -16424.357,E2 -16424.357} C_VEL
LIN {X 0,Y 307.607,Z 405.587,A -85,B 0,C 180,E1 -16425.37,E2 -16425.37} C_VEL
LIN {X 0,Y 306.022,Z 416.792,A -85,B 0,C 180,E1 -16426.632,E2 -16426.632} C_VEL
LIN {X 0,Y 304.19,Z 427.567,A -85,B 0,C 180,E1 -16428.156,E2 -16428.156} C_VEL
LIN {X 0,Y 302.495,Z 437.06,A -85,B 0,C 180,E1 -16429.854,E2 -16429.854} C_VEL
LIN {X 0,Y 300.887,Z 445.622,A -85,B 0,C 180,E1 -16431.76,E2 -16431.76} C_VEL
LIN {X 0,Y 299.541,Z 452.725,A -85,B 0,C 180,E1 -16433.729,E2 -16433.729} C_VEL
LIN {X 0,Y 298.514,Z 458.143,A -85,B 0,C 180,E1 -16435.597,E2 -16435.597} C_VEL
LIN {X 0,Y 297.63,Z 463.089,A -85,B 0,C 180,E1 -16437.755,E2 -16437.755} C_VEL
LIN {X 0,Y 296.958,Z 467.176,A -85,B 0,C 180,E1 -16440.2,E2 -16440.2} C_VEL
LIN {X 0,Y 296.62,Z 468.989,A -85,B 0,C 180,E1 -16441.716,E2 -16441.716} C_VEL
LIN {X 0,Y 296.262,Z 470.941,A -85,B 0,C 180,E1 -16444.334,E2 -16444.334} C_VEL
LIN {X 0,Y 296.113,Z 471.395,A -85,B 0,C 180,E1 -16446.206,E2 -16446.206} C_VEL
LIN {X 0,Y 296.113,Z 471.22,A -85,B 0,C 180,E1 -16447.747,E2 -16447.747} C_VEL
LIN {X 0,Y 296.177,Z 470.596,A -85,B 0,C 180,E1 -16449.151,E2 -16449.151} C_VEL
LIN {X 0,Y 296.44,Z 468.631,A -85,B 0,C 180,E1 -16451.479,E2 -16451.479} C_VEL
LIN {X 0,Y 296.76,Z 465.931,A -85,B 0,C 180,E1 -16453.491,E2 -16453.491} C_VEL
LIN {X 0,Y 297.303,Z 461.779,A -85,B 0,C 180,E1 -16455.717,E2 -16455.717} C_VEL
LIN {X 0,Y 297.979,Z 456.802,A -85,B 0,C 180,E1 -16457.746,E2 -16457.746} C_VEL
LIN {X 0,Y 298.961,Z 450.034,A -85,B 0,C 180,E1 -16459.915,E2 -16459.915} C_VEL
LIN {X 0,Y 300.206,Z 442.047,A -85,B 0,C 180,E1 -16461.927,E2 -16461.927} C_VEL
LIN {X 0,Y 301.452,Z 433.642,A -85,B 0,C 180,E1 -16463.643,E2 -16463.643} C_VEL
LIN {X 0,Y 302.885,Z 424.232,A -85,B 0,C 180,E1 -16465.205,E2 -16465.205} C_VEL
LIN {X 0,Y 304.194,Z 414.456,A -85,B 0,C 180,E1 -16466.524,E2 -16466.524} C_VEL
LIN {X 0,Y 305.52,Z 403.577,A -85,B 0,C 180,E1 -16467.694,E2 -16467.694} C_VEL
LIN {X 0,Y 306.717,Z 390.546,A -85,B 0,C 180,E1 -16468.77,E2 -16468.77} C_VEL
LIN {X 0,Y 307.68,Z 378.058,A -85,B 0,C 180,E1 -16469.51,E2 -16469.51} C_VEL
LIN {X 0,Y 308.399,Z 365.074,A -85,B 0,C 180,E1 -16470.001,E2 -16470.001} C_VEL
LIN {X 0,Y 310.072,Z 293.938,A -85,B 0,C 180,E1 -16471.698,E2 -16471.698} C_VEL
LIN {X 0,Y 306.553,Z 275.622,A -85,B 0,C 180,E1 -16472.441,E2 -16472.441} C_VEL
LIN {X 0,Y 301.126,Z 261.295,A -85,B 0,C 180,E1 -16473.275,E2 -16473.275} C_VEL
LIN {X 0,Y 300.779,Z 260.116,A -85,B 0,C 180,E1 -16473.417,E2 -16473.417} C_VEL
LIN {X 0,Y 298.773,Z 249.893,A -85,B 0,C 180,E1 -16477.01,E2 -16477.01} C_VEL
LIN {X 0,Y 298.603,Z 249.783,A -85,B 0,C 180,E1 -16479.484,E2 -16479.484} C_VEL
LIN {X 0,Y 298.52,Z 249.791,A -85,B 0,C 180,E1 -16483.618,E2 -16483.618} C_VEL
LIN {X 0,Y 298.517,Z 249.794,A -85,B 0,C 180,E1 -16486.411,E2 -16486.411} C_VEL
LIN {X 0,Y 298.467,Z 249.8,A -85,B 0,C 180,E1 -16489.65,E2 -16489.65} C_VEL
LIN {X 0,Y 298.392,Z 249.809,A -85,B 0,C 180,E1 -16493.604,E2 -16493.604} C_VEL
LIN {X 0,Y 298.38,Z 249.818,A -85,B 0,C 180,E1 -16496.586,E2 -16496.586} C_VEL
LIN {X 0,Y 298.334,Z 249.808,A -85,B 0,C 180,E1 -16499.651,E2 -16499.651} C_VEL
LIN {X 0,Y 298.366,Z 249.817,A -85,B 0,C 180,E1 -16502.805,E2 -16502.805} C_VEL
LIN {X 0,Y 298.378,Z 249.802,A -85,B 0,C 180,E1 -16506.076,E2 -16506.076} C_VEL
LIN {X 0,Y 298.351,Z 249.819,A -85,B 0,C 180,E1 -16509.496,E2 -16509.496} C_VEL
LIN {X 0,Y 298.347,Z 249.802,A -85,B 0,C 180,E1 -16513.102,E2 -16513.102} C_VEL
LIN {X 0,Y 298.35,Z 249.822,A -85,B 0,C 180,E1 -16516.919,E2 -16516.919} C_VEL
LIN {X 0,Y 298.368,Z 249.791,A -85,B 0,C 180,E1 -16521.016,E2 -16521.016} C_VEL
LIN {X 0,Y 298.38,Z 249.796,A -85,B 0,C 180,E1 -16522.735,E2 -16522.735} C_VEL
LIN {X 0,Y 297.753,Z 249.887,A -85,B 0,C 180,E1 -16523.861,E2 -16523.861} C_VEL
LIN {X 0,Y 294.912,Z 250.248,A -85,B 0,C 180,E1 -16525.695,E2 -16525.695} C_VEL
LIN {X 0,Y 292.463,Z 250.551,A -85,B 0,C 180,E1 -16527.183,E2 -16527.183} C_VEL
LIN {X 0,Y 291.391,Z 250.68,A -85,B 0,C 180,E1 -16528.337,E2 -16528.337} C_VEL
LIN {X 0,Y 291.293,Z 250.681,A -85,B 0,C 180,E1 -16528.728,E2 -16528.728} C_VEL
LIN {X 0,Y 291.318,Z 250.671,A -85,B 0,C 180,E1 -16532.724,E2 -16532.724} C_VEL
LIN {X 0,Y 291.349,Z 250.691,A -85,B 0,C 180,E1 -16536.442,E2 -16536.442} C_VEL
LIN {X 0,Y 291.434,Z 250.663,A -85,B 0,C 180,E1 -16540.274,E2 -16540.274} C_VEL
LIN {X 0,Y 291.494,Z 250.657,A -85,B 0,C 180,E1 -16544.671,E2 -16544.671} C_VEL
LIN {X 0,Y 291.526,Z 250.668,A -85,B 0,C 180,E1 -16548.885,E2 -16548.885} C_VEL
LIN {X 0,Y 291.65,Z 250.635,A -85,B 0,C 180,E1 -16551.692,E2 -16551.692} C_VEL
LIN {X 0,Y 291.597,Z 250.625,A -85,B 0,C 180,E1 -16554.473,E2 -16554.473} C_VEL
LIN {X 0,Y 291.872,Z 250.625,A -85,B 0,C 180,E1 -16558.625,E2 -16558.625} C_VEL
LIN {X 0,Y 291.88,Z 250.621,A -85,B 0,C 180,E1 -16561.384,E2 -16561.384} C_VEL
LIN {X 0,Y 291.709,Z 250.626,A -85,B 0,C 180,E1 -16566.923,E2 -16566.923} C_VEL
LIN {X 0,Y 291.575,Z 250.662,A -85,B 0,C 180,E1 -16569.718,E2 -16569.718} C_VEL
LIN {X 0,Y 291.523,Z 250.652,A -85,B 0,C 180,E1 -16573.955,E2 -16573.955} C_VEL
LIN {X 0,Y 291.449,Z 250.661,A -85,B 0,C 180,E1 -16576.824,E2 -16576.824} C_VEL
LIN {X 0,Y 291.434,Z 250.681,A -85,B 0,C 180,E1 -16579.864,E2 -16579.864} C_VEL
LIN {X 0,Y 291.37,Z 250.664,A -85,B 0,C 180,E1 -16584.212,E2 -16584.212} C_VEL
LIN {X 0,Y 291.365,Z 250.693,A -85,B 0,C 180,E1 -16587.282,E2 -16587.282} C_VEL
LIN {X 0,Y 291.33,Z 250.683,A -85,B 0,C 180,E1 -16590.442,E2 -16590.442} C_VEL
LIN {X 0,Y 291.356,Z 250.693,A -85,B 0,C 180,E1 -16593.701,E2 -16593.701} C_VEL
LIN {X 0,Y 291.365,Z 250.679,A -85,B 0,C 180,E1 -16597.25,E2 -16597.25} C_VEL
LIN {X 0,Y 291.314,Z 250.697,A -85,B 0,C 180,E1 -16600.65,E2 -16600.65} C_VEL
LIN {X 0,Y 291.296,Z 250.699,A -85,B 0,C 180,E1 -16604.405,E2 -16604.405} C_VEL
LIN {X 0,Y 291.309,Z 250.697,A -85,B 0,C 180,E1 -16608.413,E2 -16608.413} C_VEL
LIN {X 0,Y 291.347,Z 250.695,A -85,B 0,C 180,E1 -16611.156,E2 -16611.156} C_VEL
LIN {X 0,Y 291.369,Z 250.692,A -85,B 0,C 180,E1 -16614.626,E2 -16614.626} C_VEL
LIN {X 0,Y 291.385,Z 250.84,A -85,B 0,C 180,E1 -16617.37,E2 -16617.37} C_VEL
LIN {X 0,Y 293.371,Z 259.901,A -85,B 0,C 180,E1 -16620.586,E2 -16620.586} C_VEL
LIN {X 0,Y 294.928,Z 267.715,A -85,B 0,C 180,E1 -16623.153,E2 -16623.153} C_VEL
LIN {X 0,Y 297.458,Z 274.558,A -85,B 0,C 180,E1 -16623.616,E2 -16623.616} C_VEL
LIN {X 0,Y 298.732,Z 279.461,A -85,B 0,C 180,E1 -16623.855,E2 -16623.855} C_VEL
LIN {X 0,Y 303.343,Z 307.669,A -85,B 0,C 180,E1 -16624.973,E2 -16624.973} C_VEL
LIN {X 0,Y 301.575,Z 375.313,A -85,B 0,C 180,E1 -16626.625,E2 -16626.625} C_VEL
LIN {X 0,Y 300.714,Z 389.133,A -85,B 0,C 180,E1 -16627.226,E2 -16627.226} C_VEL
LIN {X 0,Y 299.563,Z 401.725,A -85,B 0,C 180,E1 -16628.042,E2 -16628.042} C_VEL
LIN {X 0,Y 298.179,Z 413.744,A -85,B 0,C 180,E1 -16629.114,E2 -16629.114} C_VEL
LIN {X 0,Y 296.662,Z 425.25,A -85,B 0,C 180,E1 -16630.449,E2 -16630.449} C_VEL
LIN {X 0,Y 295.201,Z 435.628,A -85,B 0,C 180,E1 -16631.97,E2 -16631.97} C_VEL
LIN {X 0,Y 293.822,Z 444.935,A -85,B 0,C 180,E1 -16633.676,E2 -16633.676} C_VEL
LIN {X 0,Y 292.352,Z 453.963,A -85,B 0,C 180,E1 -16635.734,E2 -16635.734} C_VEL
LIN {X 0,Y 291.17,Z 461.224,A -85,B 0,C 180,E1 -16637.806,E2 -16637.806} C_VEL
LIN {X 0,Y 290.505,Z 466.12,A -85,B 0,C 180,E1 -16639.545,E2 -16639.545} C_VEL
LIN {X 0,Y 289.919,Z 470.868,A -85,B 0,C 180,E1 -16641.636,E2 -16641.636} C_VEL
LIN {X 0,Y 289.575,Z 474.487,A -85,B 0,C 180,E1 -16643.729,E2 -16643.729} C_VEL
LIN {X 0,Y 289.406,Z 477.081,A -85,B 0,C 180,E1 -16645.821,E2 -16645.821} C_VEL
LIN {X 0,Y 289.399,Z 478.299,A -85,B 0,C 180,E1 -16647.215,E2 -16647.215} C_VEL
LIN {X 0,Y 289.38,Z 479.076,A -85,B 0,C 180,E1 -16648.607,E2 -16648.607} C_VEL
LIN {X 0,Y 289.38,Z 479.444,A -85,B 0,C 180,E1 -16649.999,E2 -16649.999} C_VEL
LIN {X 0,Y 289.379,Z 479.425,A -85,B 0,C 180,E1 -16651.39,E2 -16651.39} C_VEL
LIN {X 0,Y 289.401,Z 479.02,A -85,B 0,C 180,E1 -16652.783,E2 -16652.783} C_VEL
LIN {X 0,Y 289.418,Z 478.19,A -85,B 0,C 180,E1 -16654.176,E2 -16654.176} C_VEL
LIN {X 0,Y 289.529,Z 476.944,A -85,B 0,C 180,E1 -16655.571,E2 -16655.571} C_VEL
LIN {X 0,Y 289.834,Z 474.307,A -85,B 0,C 180,E1 -16657.663,E2 -16657.663} C_VEL
LIN {X 0,Y 290.373,Z 470.659,A -85,B 0,C 180,E1 -16659.753,E2 -16659.753} C_VEL
LIN {X 0,Y 291.218,Z 465.905,A -85,B 0,C 180,E1 -16661.836,E2 -16661.836} C_VEL
LIN {X 0,Y 292.601,Z 458.791,A -85,B 0,C 180,E1 -16664.251,E2 -16664.251} C_VEL
LIN {X 0,Y 294.218,Z 451.067,A -85,B 0,C 180,E1 -16666.299,E2 -16666.299} C_VEL
LIN {X 0,Y 295.936,Z 441.585,A -85,B 0,C 180,E1 -16668.303,E2 -16668.303} C_VEL
LIN {X 0,Y 297.74,Z 431.448,A -85,B 0,C 180,E1 -16670.014,E2 -16670.014} C_VEL
LIN {X 0,Y 299.733,Z 420.2,A -85,B 0,C 180,E1 -16671.49,E2 -16671.49} C_VEL
LIN {X 0,Y 301.274,Z 409.22,A -85,B 0,C 180,E1 -16672.636,E2 -16672.636} C_VEL
LIN {X 0,Y 302.834,Z 397.075,A -85,B 0,C 180,E1 -16673.597,E2 -16673.597} C_VEL
LIN {X 0,Y 303.97,Z 384.417,A -85,B 0,C 180,E1 -16674.319,E2 -16674.319} C_VEL
LIN {X 0,Y 304.852,Z 370.681,A -85,B 0,C 180,E1 -16674.806,E2 -16674.806} C_VEL
LIN {X 0,Y 306.563,Z 308.576,A -85,B 0,C 180,E1 -16676.327,E2 -16676.327} C_VEL
LIN {X 0,Y 303.395,Z 289.716,A -85,B 0,C 180,E1 -16677.184,E2 -16677.184} C_VEL
LIN {X 0,Y 301.83,Z 282.501,A -85,B 0,C 180,E1 -16677.559,E2 -16677.559} C_VEL
LIN {X 0,Y 296.719,Z 270.532,A -85,B 0,C 180,E1 -16678.488,E2 -16678.488} C_VEL
LIN {X 0,Y 295.26,Z 267.057,A -85,B 0,C 180,E1 -16678.829,E2 -16678.829} C_VEL
LIN {X 0,Y 293.322,Z 258.535,A -85,B 0,C 180,E1 -16681.809,E2 -16681.809} C_VEL
LIN {X 0,Y 291.402,Z 250.838,A -85,B 0,C 180,E1 -16684.777,E2 -16684.777} C_VEL
LIN {X 0,Y 291.366,Z 250.683,A -85,B 0,C 180,E1 -16687.246,E2 -16687.246} C_VEL
LIN {X 0,Y 291.307,Z 250.687,A -85,B 0,C 180,E1 -16690.645,E2 -16690.645} C_VEL
LIN {X 0,Y 291.288,Z 250.703,A -85,B 0,C 180,E1 -16694.4,E2 -16694.4} C_VEL
LIN {X 0,Y 291.3,Z 250.695,A -85,B 0,C 180,E1 -16698.408,E2 -16698.408} C_VEL
LIN {X 0,Y 291.337,Z 250.688,A -85,B 0,C 180,E1 -16701.151,E2 -16701.151} C_VEL
LIN {X 0,Y 291.358,Z 250.686,A -85,B 0,C 180,E1 -16704.621,E2 -16704.621} C_VEL
LIN {X 0,Y 291.368,Z 250.686,A -85,B 0,C 180,E1 -16707.946,E2 -16707.946} C_VEL
LIN {X 0,Y 291.344,Z 250.692,A -85,B 0,C 180,E1 -16711.15,E2 -16711.15} C_VEL
LIN {X 0,Y 291.358,Z 250.689,A -85,B 0,C 180,E1 -16714.262,E2 -16714.262} C_VEL
LIN {X 0,Y 291.365,Z 250.681,A -85,B 0,C 180,E1 -16717.294,E2 -16717.294} C_VEL
LIN {X 0,Y 291.458,Z 250.678,A -85,B 0,C 180,E1 -16720.266,E2 -16720.266} C_VEL
LIN {X 0,Y 291.496,Z 250.676,A -85,B 0,C 180,E1 -16724.661,E2 -16724.661} C_VEL
LIN {X 0,Y 291.524,Z 250.671,A -85,B 0,C 180,E1 -16728.876,E2 -16728.876} C_VEL
LIN {X 0,Y 291.658,Z 250.643,A -85,B 0,C 180,E1 -16731.683,E2 -16731.683} C_VEL
LIN {X 0,Y 291.594,Z 250.661,A -85,B 0,C 180,E1 -16734.463,E2 -16734.463} C_VEL
LIN {X 0,Y 291.869,Z 250.627,A -85,B 0,C 180,E1 -16738.616,E2 -16738.616} C_VEL
LIN {X 0,Y 291.856,Z 250.619,A -85,B 0,C 180,E1 -16741.375,E2 -16741.375} C_VEL
LIN {X 0,Y 291.673,Z 250.65,A -85,B 0,C 180,E1 -16746.915,E2 -16746.915} C_VEL
LIN {X 0,Y 291.555,Z 250.66,A -85,B 0,C 180,E1 -16749.709,E2 -16749.709} C_VEL
LIN {X 0,Y 291.5,Z 250.669,A -85,B 0,C 180,E1 -16753.946,E2 -16753.946} C_VEL
LIN {X 0,Y 291.427,Z 250.677,A -85,B 0,C 180,E1 -16756.816,E2 -16756.816} C_VEL
LIN {X 0,Y 291.407,Z 250.683,A -85,B 0,C 180,E1 -16759.855,E2 -16759.855} C_VEL
LIN {X 0,Y 291.345,Z 250.696,A -85,B 0,C 180,E1 -16764.204,E2 -16764.204} C_VEL
LIN {X 0,Y 291.333,Z 250.693,A -85,B 0,C 180,E1 -16767.274,E2 -16767.274} C_VEL
LIN {X 0,Y 291.297,Z 250.702,A -85,B 0,C 180,E1 -16770.435,E2 -16770.435} C_VEL
LIN {X 0,Y 291.382,Z 250.808,A -85,B 0,C 180,E1 -16774.466,E2 -16774.466} C_VEL
LIN {X 0,Y 293.566,Z 259.563,A -85,B 0,C 180,E1 -16777.815,E2 -16777.815} C_VEL
LIN {X 0,Y 293.886,Z 260.761,A -85,B 0,C 180,E1 -16778.101,E2 -16778.101} C_VEL
LIN {X 0,Y 300.928,Z 275.886,A -85,B 0,C 180,E1 -16779.395,E2 -16779.395} C_VEL
LIN {X 0,Y 304.96,Z 286.157,A -85,B 0,C 180,E1 -16780.13,E2 -16780.13} C_VEL
LIN {X 0,Y 306.969,Z 297.243,A -85,B 0,C 180,E1 -16780.648,E2 -16780.648} C_VEL
LIN {X 0,Y 304.66,Z 368.427,A -85,B 0,C 180,E1 -16782.393,E2 -16782.393} C_VEL
LIN {X 0,Y 303.694,Z 381.988,A -85,B 0,C 180,E1 -16782.99,E2 -16782.99} C_VEL
LIN {X 0,Y 302.554,Z 394.487,A -85,B 0,C 180,E1 -16783.82,E2 -16783.82} C_VEL
LIN {X 0,Y 301.016,Z 406.483,A -85,B 0,C 180,E1 -16784.898,E2 -16784.898} C_VEL
LIN {X 0,Y 299.403,Z 417.465,A -85,B 0,C 180,E1 -16786.177,E2 -16786.177} C_VEL
LIN {X 0,Y 297.526,Z 427.863,A -85,B 0,C 180,E1 -16787.686,E2 -16787.686} C_VEL
LIN {X 0,Y 295.686,Z 437.723,A -85,B 0,C 180,E1 -16789.507,E2 -16789.507} C_VEL
LIN {X 0,Y 293.924,Z 446.606,A -85,B 0,C 180,E1 -16791.563,E2 -16791.563} C_VEL
LIN {X 0,Y 292.559,Z 453.368,A -85,B 0,C 180,E1 -16793.521,E2 -16793.521} C_VEL
LIN {X 0,Y 291.414,Z 459.154,A -85,B 0,C 180,E1 -16795.626,E2 -16795.626} C_VEL
LIN {X 0,Y 290.507,Z 463.88,A -85,B 0,C 180,E1 -16797.846,E2 -16797.846} C_VEL
LIN {X 0,Y 290.083,Z 466.482,A -85,B 0,C 180,E1 -16799.419,E2 -16799.419} C_VEL
LIN {X 0,Y 289.714,Z 468.514,A -85,B 0,C 180,E1 -16800.978,E2 -16800.978} C_VEL
LIN {X 0,Y 289.366,Z 469.974,A -85,B 0,C 180,E1 -16802.52,E2 -16802.52} C_VEL
LIN {X 0,Y 289.178,Z 470.969,A -85,B 0,C 180,E1 -16804.06,E2 -16804.06} C_VEL
LIN {X 0,Y 289.04,Z 471.435,A -85,B 0,C 180,E1 -16805.586,E2 -16805.586} C_VEL
LIN {X 0,Y 289.01,Z 471.381,A -85,B 0,C 180,E1 -16807.51,E2 -16807.51} C_VEL
LIN {X 0,Y 289.158,Z 470.051,A -85,B 0,C 180,E1 -16810.108,E2 -16810.108} C_VEL
LIN {X 0,Y 289.365,Z 468.662,A -85,B 0,C 180,E1 -16811.596,E2 -16811.596} C_VEL
LIN {X 0,Y 289.727,Z 465.705,A -85,B 0,C 180,E1 -16813.803,E2 -16813.803} C_VEL
LIN {X 0,Y 290.291,Z 461.634,A -85,B 0,C 180,E1 -16815.991,E2 -16815.991} C_VEL
LIN {X 0,Y 291.054,Z 456.352,A -85,B 0,C 180,E1 -16818.157,E2 -16818.157} C_VEL
LIN {X 0,Y 292.142,Z 449.039,A -85,B 0,C 180,E1 -16820.475,E2 -16820.475} C_VEL
LIN {X 0,Y 293.417,Z 441.258,A -85,B 0,C 180,E1 -16822.431,E2 -16822.431} C_VEL
LIN {X 0,Y 294.775,Z 432.665,A -85,B 0,C 180,E1 -16824.186,E2 -16824.186} C_VEL
LIN {X 0,Y 296.243,Z 423.237,A -85,B 0,C 180,E1 -16825.745,E2 -16825.745} C_VEL
LIN {X 0,Y 297.678,Z 412.862,A -85,B 0,C 180,E1 -16827.125,E2 -16827.125} C_VEL
LIN {X 0,Y 299.025,Z 401.578,A -85,B 0,C 180,E1 -16828.318,E2 -16828.318} C_VEL
LIN {X 0,Y 300.19,Z 389.103,A -85,B 0,C 180,E1 -16829.33,E2 -16829.33} C_VEL
LIN {X 0,Y 301.154,Z 376.58,A -85,B 0,C 180,E1 -16830.045,E2 -16830.045} C_VEL
LIN {X 0,Y 301.802,Z 363.417,A -85,B 0,C 180,E1 -16830.527,E2 -16830.527} C_VEL
LIN {X 0,Y 303.533,Z 295.051,A -85,B 0,C 180,E1 -16832.179,E2 -16832.179} C_VEL
LIN {X 0,Y 300.184,Z 277.714,A -85,B 0,C 180,E1 -16832.903,E2 -16832.903} C_VEL
LIN {X 0,Y 294.569,Z 263.115,A -85,B 0,C 180,E1 -16833.772,E2 -16833.772} C_VEL
LIN {X 0,Y 293.529,Z 260.239,A -85,B 0,C 180,E1 -16834.043,E2 -16834.043} C_VEL
LIN {X 0,Y 291.764,Z 250.955,A -85,B 0,C 180,E1 -16837.353,E2 -16837.353} C_VEL
LIN {X 0,Y 291.71,Z 250.66,A -85,B 0,C 180,E1 -16837.616,E2 -16837.616} C_VEL
LIN {X 0,Y 291.504,Z 250.676,A -85,B 0,C 180,E1 -16841.122,E2 -16841.122} C_VEL
LIN {X 0,Y 291.508,Z 250.673,A -85,B 0,C 180,E1 -16845.38,E2 -16845.38} C_VEL
LIN {X 0,Y 291.422,Z 250.677,A -85,B 0,C 180,E1 -16849.878,E2 -16849.878} C_VEL
LIN {X 0,Y 291.331,Z 250.686,A -85,B 0,C 180,E1 -16854.212,E2 -16854.212} C_VEL
LIN {X 0,Y 291.324,Z 250.695,A -85,B 0,C 180,E1 -16857.282,E2 -16857.282} C_VEL
LIN {X 0,Y 291.277,Z 250.694,A -85,B 0,C 180,E1 -16860.445,E2 -16860.445} C_VEL
LIN {X 0,Y 291.318,Z 250.692,A -85,B 0,C 180,E1 -16863.703,E2 -16863.703} C_VEL
LIN {X 0,Y 291.328,Z 250.693,A -85,B 0,C 180,E1 -16867.252,E2 -16867.252} C_VEL
LIN {X 0,Y 291.277,Z 250.693,A -85,B 0,C 180,E1 -16870.653,E2 -16870.653} C_VEL
LIN {X 0,Y 291.261,Z 250.692,A -85,B 0,C 180,E1 -16874.409,E2 -16874.409} C_VEL
LIN {X 0,Y 291.275,Z 250.698,A -85,B 0,C 180,E1 -16878.417,E2 -16878.417} C_VEL
LIN {X 0,Y 291.316,Z 250.669,A -85,B 0,C 180,E1 -16881.16,E2 -16881.16} C_VEL
LIN {X 0,Y 291.34,Z 250.688,A -85,B 0,C 180,E1 -16884.63,E2 -16884.63} C_VEL
LIN {X 0,Y 291.293,Z 250.681,A -85,B 0,C 180,E1 -16888.728,E2 -16888.728} C_VEL
LIN {X 0,Y 290.595,Z 250.763,A -85,B 0,C 180,E1 -16889.882,E2 -16889.882} C_VEL
LIN {X 0,Y 287.726,Z 251.113,A -85,B 0,C 180,E1 -16891.763,E2 -16891.763} C_VEL
LIN {X 0,Y 285.329,Z 251.421,A -85,B 0,C 180,E1 -16893.29,E2 -16893.29} C_VEL
LIN {X 0,Y 284.331,Z 251.558,A -85,B 0,C 180,E1 -16894.473,E2 -16894.473} C_VEL
LIN {X 0,Y 284.265,Z 251.565,A -85,B 0,C 180,E1 -16894.873,E2 -16894.873} C_VEL
LIN {X 0,Y 284.296,Z 251.566,A -85,B 0,C 180,E1 -16898.24,E2 -16898.24} C_VEL
LIN {X 0,Y 284.356,Z 251.53,A -85,B 0,C 180,E1 -16901.264,E2 -16901.264} C_VEL
LIN {X 0,Y 284.459,Z 251.538,A -85,B 0,C 180,E1 -16905.702,E2 -16905.702} C_VEL
LIN {X 0,Y 284.513,Z 251.537,A -85,B 0,C 180,E1 -16910.048,E2 -16910.048} C_VEL
LIN {X 0,Y 284.641,Z 251.496,A -85,B 0,C 180,E1 -16912.914,E2 -16912.914} C_VEL
LIN {X 0,Y 284.84,Z 251.502,A -85,B 0,C 180,E1 -16918.591,E2 -16918.591} C_VEL
LIN {X 0,Y 284.846,Z 251.497,A -85,B 0,C 180,E1 -16921.419,E2 -16921.419} C_VEL
LIN {X 0,Y 284.664,Z 251.506,A -85,B 0,C 180,E1 -16927.096,E2 -16927.096} C_VEL
LIN {X 0,Y 284.521,Z 251.542,A -85,B 0,C 180,E1 -16929.961,E2 -16929.961} C_VEL
LIN {X 0,Y 284.471,Z 251.525,A -85,B 0,C 180,E1 -16934.308,E2 -16934.308} C_VEL
LIN {X 0,Y 284.384,Z 251.558,A -85,B 0,C 180,E1 -16938.744,E2 -16938.744} C_VEL
LIN {X 0,Y 284.322,Z 251.561,A -85,B 0,C 180,E1 -16941.768,E2 -16941.768} C_VEL
LIN {X 0,Y 284.317,Z 251.546,A -85,B 0,C 180,E1 -16944.853,E2 -16944.853} C_VEL
LIN {X 0,Y 284.295,Z 251.57,A -85,B 0,C 180,E1 -16948.019,E2 -16948.019} C_VEL
LIN {X 0,Y 284.297,Z 251.555,A -85,B 0,C 180,E1 -16951.279,E2 -16951.279} C_VEL
LIN {X 0,Y 284.349,Z 251.564,A -85,B 0,C 180,E1 -16955.349,E2 -16955.349} C_VEL
LIN {X 0,Y 284.308,Z 251.561,A -85,B 0,C 180,E1 -16958.174,E2 -16958.174} C_VEL
LIN {X 0,Y 284.25,Z 251.566,A -85,B 0,C 180,E1 -16962.119,E2 -16962.119} C_VEL
LIN {X 0,Y 284.251,Z 251.571,A -85,B 0,C 180,E1 -16966.187,E2 -16966.187} C_VEL
LIN {X 0,Y 284.298,Z 251.57,A -85,B 0,C 180,E1 -16970.031,E2 -16970.031} C_VEL
LIN {X 0,Y 284.333,Z 251.567,A -85,B 0,C 180,E1 -16973.613,E2 -16973.613} C_VEL
LIN {X 0,Y 284.338,Z 251.667,A -85,B 0,C 180,E1 -16976.847,E2 -16976.847} C_VEL
LIN {X 0,Y 285.859,Z 258.423,A -85,B 0,C 180,E1 -16979.378,E2 -16979.378} C_VEL
LIN {X 0,Y 287.706,Z 267.65,A -85,B 0,C 180,E1 -16982.51,E2 -16982.51} C_VEL
LIN {X 0,Y 290.39,Z 274.829,A -85,B 0,C 180,E1 -16983.005,E2 -16983.005} C_VEL
LIN {X 0,Y 292.096,Z 279.77,A -85,B 0,C 180,E1 -16983.291,E2 -16983.291} C_VEL
LIN {X 0,Y 296.817,Z 308.878,A -85,B 0,C 180,E1 -16984.479,E2 -16984.479} C_VEL
LIN {X 0,Y 294.946,Z 375.689,A -85,B 0,C 180,E1 -16986.15,E2 -16986.15} C_VEL
LIN {X 0,Y 294.044,Z 389.525,A -85,B 0,C 180,E1 -16986.772,E2 -16986.772} C_VEL
LIN {X 0,Y 292.858,Z 401.982,A -85,B 0,C 180,E1 -16987.605,E2 -16987.605} C_VEL
LIN {X 0,Y 291.549,Z 413.116,A -85,B 0,C 180,E1 -16988.616,E2 -16988.616} C_VEL
LIN {X 0,Y 289.977,Z 424.722,A -85,B 0,C 180,E1 -16989.979,E2 -16989.979} C_VEL
LIN {X 0,Y 288.399,Z 435.174,A -85,B 0,C 180,E1 -16991.53,E2 -16991.53} C_VEL
LIN {X 0,Y 286.99,Z 444.566,A -85,B 0,C 180,E1 -16993.276,E2 -16993.276} C_VEL
LIN {X 0,Y 285.454,Z 453.64,A -85,B 0,C 180,E1 -16995.382,E2 -16995.382} C_VEL
LIN {X 0,Y 284.196,Z 460.942,A -85,B 0,C 180,E1 -16997.502,E2 -16997.502} C_VEL
LIN {X 0,Y 283.513,Z 465.873,A -85,B 0,C 180,E1 -16999.284,E2 -16999.284} C_VEL
LIN {X 0,Y 282.885,Z 470.654,A -85,B 0,C 180,E1 -17001.426,E2 -17001.426} C_VEL
LIN {X 0,Y 282.507,Z 474.302,A -85,B 0,C 180,E1 -17003.571,E2 -17003.571} C_VEL
LIN {X 0,Y 282.317,Z 476.924,A -85,B 0,C 180,E1 -17005.716,E2 -17005.716} C_VEL
LIN {X 0,Y 282.309,Z 478.156,A -85,B 0,C 180,E1 -17007.145,E2 -17007.145} C_VEL
LIN {X 0,Y 282.304,Z 478.959,A -85,B 0,C 180,E1 -17008.572,E2 -17008.572} C_VEL
LIN {X 0,Y 282.303,Z 479.339,A -85,B 0,C 180,E1 -17009.999,E2 -17009.999} C_VEL
LIN {X 0,Y 282.304,Z 479.332,A -85,B 0,C 180,E1 -17011.425,E2 -17011.425} C_VEL
LIN {X 0,Y 282.312,Z 478.94,A -85,B 0,C 180,E1 -17012.853,E2 -17012.853} C_VEL
LIN {X 0,Y 282.436,Z 477.116,A -85,B 0,C 180,E1 -17015.503,E2 -17015.503} C_VEL
LIN {X 0,Y 282.774,Z 474.295,A -85,B 0,C 180,E1 -17017.855,E2 -17017.855} C_VEL
LIN {X 0,Y 283.363,Z 470.681,A -85,B 0,C 180,E1 -17019.997,E2 -17019.997} C_VEL
LIN {X 0,Y 284.262,Z 465.966,A -85,B 0,C 180,E1 -17022.13,E2 -17022.13} C_VEL
LIN {X 0,Y 285.731,Z 458.89,A -85,B 0,C 180,E1 -17024.601,E2 -17024.601} C_VEL
LIN {X 0,Y 287.396,Z 451.228,A -85,B 0,C 180,E1 -17026.697,E2 -17026.697} C_VEL
LIN {X 0,Y 288.887,Z 443.401,A -85,B 0,C 180,E1 -17028.436,E2 -17028.436} C_VEL
LIN {X 0,Y 290.895,Z 432.793,A -85,B 0,C 180,E1 -17030.321,E2 -17030.321} C_VEL
LIN {X 0,Y 292.938,Z 421.998,A -85,B 0,C 180,E1 -17031.829,E2 -17031.829} C_VEL
LIN {X 0,Y 294.773,Z 409.735,A -85,B 0,C 180,E1 -17033.164,E2 -17033.164} C_VEL
LIN {X 0,Y 296.357,Z 397.763,A -85,B 0,C 180,E1 -17034.145,E2 -17034.145} C_VEL
LIN {X 0,Y 297.636,Z 384.692,A -85,B 0,C 180,E1 -17034.918,E2 -17034.918} C_VEL
LIN {X 0,Y 298.526,Z 371.318,A -85,B 0,C 180,E1 -17035.413,E2 -17035.413} C_VEL
LIN {X 0,Y 300.376,Z 309.596,A -85,B 0,C 180,E1 -17036.956,E2 -17036.956} C_VEL
LIN {X 0,Y 296.924,Z 288.947,A -85,B 0,C 180,E1 -17037.933,E2 -17037.933} C_VEL
LIN {X 0,Y 295.931,Z 285.1,A -85,B 0,C 180,E1 -17038.159,E2 -17038.159} C_VEL
LIN {X 0,Y 291.07,Z 273.706,A -85,B 0,C 180,E1 -17039.084,E2 -17039.084} C_VEL
LIN {X 0,Y 288.079,Z 266.982,A -85,B 0,C 180,E1 -17039.718,E2 -17039.718} C_VEL
LIN {X 0,Y 285.82,Z 257.296,A -85,B 0,C 180,E1 -17043.272,E2 -17043.272} C_VEL
LIN {X 0,Y 284.35,Z 251.791,A -85,B 0,C 180,E1 -17045.502,E2 -17045.502} C_VEL
LIN {X 0,Y 284.305,Z 251.572,A -85,B 0,C 180,E1 -17048.168,E2 -17048.168} C_VEL
LIN {X 0,Y 284.244,Z 251.58,A -85,B 0,C 180,E1 -17052.114,E2 -17052.114} C_VEL
LIN {X 0,Y 284.243,Z 251.576,A -85,B 0,C 180,E1 -17056.182,E2 -17056.182} C_VEL
LIN {X 0,Y 284.288,Z 251.574,A -85,B 0,C 180,E1 -17060.026,E2 -17060.026} C_VEL
LIN {X 0,Y 284.322,Z 251.568,A -85,B 0,C 180,E1 -17063.608,E2 -17063.608} C_VEL
LIN {X 0,Y 284.309,Z 251.569,A -85,B 0,C 180,E1 -17067.186,E2 -17067.186} C_VEL
LIN {X 0,Y 284.338,Z 251.566,A -85,B 0,C 180,E1 -17070.369,E2 -17070.369} C_VEL
LIN {X 0,Y 284.305,Z 251.565,A -85,B 0,C 180,E1 -17073.575,E2 -17073.575} C_VEL
LIN {X 0,Y 284.328,Z 251.558,A -85,B 0,C 180,E1 -17076.699,E2 -17076.699} C_VEL
LIN {X 0,Y 284.376,Z 251.56,A -85,B 0,C 180,E1 -17079.9,E2 -17079.9} C_VEL
LIN {X 0,Y 284.446,Z 251.553,A -85,B 0,C 180,E1 -17084.487,E2 -17084.487} C_VEL
LIN {X 0,Y 284.478,Z 251.547,A -85,B 0,C 180,E1 -17088.597,E2 -17088.597} C_VEL
LIN {X 0,Y 284.613,Z 251.52,A -85,B 0,C 180,E1 -17091.475,E2 -17091.475} C_VEL
LIN {X 0,Y 284.565,Z 251.537,A -85,B 0,C 180,E1 -17094.326,E2 -17094.326} C_VEL
LIN {X 0,Y 284.835,Z 251.504,A -85,B 0,C 180,E1 -17098.581,E2 -17098.581} C_VEL
LIN {X 0,Y 284.823,Z 251.495,A -85,B 0,C 180,E1 -17101.409,E2 -17101.409} C_VEL
LIN {X 0,Y 284.628,Z 251.528,A -85,B 0,C 180,E1 -17107.087,E2 -17107.087} C_VEL
LIN {X 0,Y 284.501,Z 251.539,A -85,B 0,C 180,E1 -17109.952,E2 -17109.952} C_VEL
LIN {X 0,Y 284.453,Z 251.549,A -85,B 0,C 180,E1 -17114.299,E2 -17114.299} C_VEL
LIN {X 0,Y 284.367,Z 251.564,A -85,B 0,C 180,E1 -17118.735,E2 -17118.735} C_VEL
LIN {X 0,Y 284.298,Z 251.573,A -85,B 0,C 180,E1 -17121.759,E2 -17121.759} C_VEL
LIN {X 0,Y 284.289,Z 251.571,A -85,B 0,C 180,E1 -17124.845,E2 -17124.845} C_VEL
LIN {X 0,Y 284.263,Z 251.565,A -85,B 0,C 180,E1 -17128.011,E2 -17128.011} C_VEL
LIN {X 0,Y 284.263,Z 251.572,A -85,B 0,C 180,E1 -17131.271,E2 -17131.271} C_VEL
LIN {X 0,Y 284.311,Z 251.672,A -85,B 0,C 180,E1 -17133.679,E2 -17133.679} C_VEL
LIN {X 0,Y 286.415,Z 259.837,A -85,B 0,C 180,E1 -17136.947,E2 -17136.947} C_VEL
LIN {X 0,Y 286.811,Z 261.135,A -85,B 0,C 180,E1 -17137.217,E2 -17137.217} C_VEL
LIN {X 0,Y 293.489,Z 274.994,A -85,B 0,C 180,E1 -17138.499,E2 -17138.499} C_VEL
LIN {X 0,Y 298.921,Z 287.951,A -85,B 0,C 180,E1 -17139.51,E2 -17139.51} C_VEL
LIN {X 0,Y 300.768,Z 298.372,A -85,B 0,C 180,E1 -17140.013,E2 -17140.013} C_VEL
LIN {X 0,Y 298.407,Z 368.314,A -85,B 0,C 180,E1 -17141.763,E2 -17141.763} C_VEL
LIN {X 0,Y 297.372,Z 381.836,A -85,B 0,C 180,E1 -17142.362,E2 -17142.362} C_VEL
LIN {X 0,Y 296.145,Z 394.899,A -85,B 0,C 180,E1 -17143.25,E2 -17143.25} C_VEL
LIN {X 0,Y 294.597,Z 406.397,A -85,B 0,C 180,E1 -17144.302,E2 -17144.302} C_VEL
LIN {X 0,Y 292.828,Z 417.796,A -85,B 0,C 180,E1 -17145.654,E2 -17145.654} C_VEL
LIN {X 0,Y 290.879,Z 428.215,A -85,B 0,C 180,E1 -17147.206,E2 -17147.206} C_VEL
LIN {X 0,Y 289.027,Z 437.568,A -85,B 0,C 180,E1 -17148.966,E2 -17148.966} C_VEL
LIN {X 0,Y 287.364,Z 445.688,A -85,B 0,C 180,E1 -17150.859,E2 -17150.859} C_VEL
LIN {X 0,Y 285.805,Z 452.937,A -85,B 0,C 180,E1 -17152.956,E2 -17152.956} C_VEL
LIN {X 0,Y 284.434,Z 459.463,A -85,B 0,C 180,E1 -17155.37,E2 -17155.37} C_VEL
LIN {X 0,Y 283.564,Z 463.734,A -85,B 0,C 180,E1 -17157.411,E2 -17157.411} C_VEL
LIN {X 0,Y 283.011,Z 466.925,A -85,B 0,C 180,E1 -17159.399,E2 -17159.399} C_VEL
LIN {X 0,Y 282.406,Z 469.631,A -85,B 0,C 180,E1 -17161.783,E2 -17161.783} C_VEL
LIN {X 0,Y 282.103,Z 470.961,A -85,B 0,C 180,E1 -17163.734,E2 -17163.734} C_VEL
LIN {X 0,Y 281.918,Z 471.601,A -85,B 0,C 180,E1 -17166.494,E2 -17166.494} C_VEL
LIN {X 0,Y 281.915,Z 471.289,A -85,B 0,C 180,E1 -17168.042,E2 -17168.042} C_VEL
LIN {X 0,Y 281.997,Z 470.544,A -85,B 0,C 180,E1 -17169.581,E2 -17169.581} C_VEL
LIN {X 0,Y 282.2,Z 469.299,A -85,B 0,C 180,E1 -17171.129,E2 -17171.129} C_VEL
LIN {X 0,Y 282.536,Z 466.61,A -85,B 0,C 180,E1 -17173.379,E2 -17173.379} C_VEL
LIN {X 0,Y 283.097,Z 462.798,A -85,B 0,C 180,E1 -17175.627,E2 -17175.627} C_VEL
LIN {X 0,Y 283.832,Z 457.797,A -85,B 0,C 180,E1 -17177.851,E2 -17177.851} C_VEL
LIN {X 0,Y 284.787,Z 451.473,A -85,B 0,C 180,E1 -17180.054,E2 -17180.054} C_VEL
LIN {X 0,Y 286.166,Z 443.538,A -85,B 0,C 180,E1 -17182.238,E2 -17182.238} C_VEL
LIN {X 0,Y 287.476,Z 435.385,A -85,B 0,C 180,E1 -17184.037,E2 -17184.037} C_VEL
LIN {X 0,Y 289.082,Z 425.377,A -85,B 0,C 180,E1 -17185.819,E2 -17185.819} C_VEL
LIN {X 0,Y 290.749,Z 414.185,A -85,B 0,C 180,E1 -17187.403,E2 -17187.403} C_VEL
LIN {X 0,Y 292.149,Z 403.175,A -85,B 0,C 180,E1 -17188.623,E2 -17188.623} C_VEL
LIN {X 0,Y 293.349,Z 391.113,A -85,B 0,C 180,E1 -17189.658,E2 -17189.658} C_VEL
LIN {X 0,Y 294.423,Z 378.103,A -85,B 0,C 180,E1 -17190.464,E2 -17190.464} C_VEL
LIN {X 0,Y 295.164,Z 365.106,A -85,B 0,C 180,E1 -17190.973,E2 -17190.973} C_VEL
LIN {X 0,Y 296.973,Z 295.861,A -85,B 0,C 180,E1 -17192.69,E2 -17192.69} C_VEL
LIN {X 0,Y 293.977,Z 280.21,A -85,B 0,C 180,E1 -17193.362,E2 -17193.362} C_VEL
LIN {X 0,Y 288.436,Z 265.853,A -85,B 0,C 180,E1 -17194.249,E2 -17194.249} C_VEL
LIN {X 0,Y 286.434,Z 260.767,A -85,B 0,C 180,E1 -17194.619,E2 -17194.619} C_VEL
LIN {X 0,Y 285.842,Z 257.614,A -85,B 0,C 180,E1 -17195.645,E2 -17195.645} C_VEL
LIN {X 0,Y 284.641,Z 251.581,A -85,B 0,C 180,E1 -17197.984,E2 -17197.984} C_VEL
LIN {X 0,Y 284.445,Z 251.54,A -85,B 0,C 180,E1 -17202.849,E2 -17202.849} C_VEL
LIN {X 0,Y 284.451,Z 251.548,A -85,B 0,C 180,E1 -17205.771,E2 -17205.771} C_VEL
LIN {X 0,Y 284.347,Z 251.559,A -85,B 0,C 180,E1 -17210.246,E2 -17210.246} C_VEL
LIN {X 0,Y 284.292,Z 251.563,A -85,B 0,C 180,E1 -17213.856,E2 -17213.856} C_VEL
LIN {X 0,Y 284.246,Z 251.57,A -85,B 0,C 180,E1 -17218.021,E2 -17218.021} C_VEL
LIN {X 0,Y 284.252,Z 251.575,A -85,B 0,C 180,E1 -17221.281,E2 -17221.281} C_VEL
LIN {X 0,Y 284.312,Z 251.55,A -85,B 0,C 180,E1 -17225.351,E2 -17225.351} C_VEL
LIN {X 0,Y 284.272,Z 251.574,A -85,B 0,C 180,E1 -17228.176,E2 -17228.176} C_VEL
LIN {X 0,Y 284.214,Z 251.561,A -85,B 0,C 180,E1 -17232.121,E2 -17232.121} C_VEL
LIN {X 0,Y 284.218,Z 251.58,A -85,B 0,C 180,E1 -17236.191,E2 -17236.191} C_VEL
LIN {X 0,Y 284.266,Z 251.555,A -85,B 0,C 180,E1 -17240.035,E2 -17240.035} C_VEL
LIN {X 0,Y 284.303,Z 251.56,A -85,B 0,C 180,E1 -17243.617,E2 -17243.617} C_VEL
LIN {X 0,Y 284.293,Z 251.569,A -85,B 0,C 180,E1 -17247.196,E2 -17247.196} C_VEL
LIN {X 0,Y 284.297,Z 251.541,A -85,B 0,C 180,E1 -17250.376,E2 -17250.376} C_VEL
LIN {X 0,Y 284.286,Z 251.554,A -85,B 0,C 180,E1 -17253.584,E2 -17253.584} C_VEL
LIN {X 0,Y 284.265,Z 251.565,A -85,B 0,C 180,E1 -17254.873,E2 -17254.873} C_VEL
LIN {X 0,Y 283.646,Z 251.654,A -85,B 0,C 180,E1 -17256.056,E2 -17256.056} C_VEL
LIN {X 0,Y 280.844,Z 252.003,A -85,B 0,C 180,E1 -17257.983,E2 -17257.983} C_VEL
LIN {X 0,Y 278.433,Z 252.289,A -85,B 0,C 180,E1 -17259.548,E2 -17259.548} C_VEL
LIN {X 0,Y 277.384,Z 252.406,A -85,B 0,C 180,E1 -17260.76,E2 -17260.76} C_VEL
LIN {X 0,Y 277.293,Z 252.41,A -85,B 0,C 180,E1 -17261.171,E2 -17261.171} C_VEL
LIN {X 0,Y 277.406,Z 252.413,A -85,B 0,C 180,E1 -17265.33,E2 -17265.33} C_VEL
LIN {X 0,Y 277.456,Z 252.419,A -85,B 0,C 180,E1 -17269.792,E2 -17269.792} C_VEL
LIN {X 0,Y 277.599,Z 252.375,A -85,B 0,C 180,E1 -17272.733,E2 -17272.733} C_VEL
LIN {X 0,Y 277.807,Z 252.378,A -85,B 0,C 180,E1 -17278.555,E2 -17278.555} C_VEL
LIN {X 0,Y 277.812,Z 252.373,A -85,B 0,C 180,E1 -17281.454,E2 -17281.454} C_VEL
LIN {X 0,Y 277.621,Z 252.385,A -85,B 0,C 180,E1 -17287.276,E2 -17287.276} C_VEL
LIN {X 0,Y 277.465,Z 252.423,A -85,B 0,C 180,E1 -17290.218,E2 -17290.218} C_VEL
LIN {X 0,Y 277.418,Z 252.4,A -85,B 0,C 180,E1 -17294.68,E2 -17294.68} C_VEL
LIN {X 0,Y 277.334,Z 252.44,A -85,B 0,C 180,E1 -17299.239,E2 -17299.239} C_VEL
LIN {X 0,Y 277.293,Z 252.417,A -85,B 0,C 180,E1 -17303.928,E2 -17303.928} C_VEL
LIN {X 0,Y 277.282,Z 252.446,A -85,B 0,C 180,E1 -17307.486,E2 -17307.486} C_VEL
LIN {X 0,Y 277.261,Z 252.435,A -85,B 0,C 180,E1 -17310.476,E2 -17310.476} C_VEL
LIN {X 0,Y 277.259,Z 252.449,A -85,B 0,C 180,E1 -17313.899,E2 -17313.899} C_VEL
LIN {X 0,Y 277.264,Z 252.435,A -85,B 0,C 180,E1 -17317.475,E2 -17317.475} C_VEL
LIN {X 0,Y 277.198,Z 252.452,A -85,B 0,C 180,E1 -17321.244,E2 -17321.244} C_VEL
LIN {X 0,Y 277.188,Z 252.458,A -85,B 0,C 180,E1 -17325.234,E2 -17325.234} C_VEL
LIN {X 0,Y 277.198,Z 252.454,A -85,B 0,C 180,E1 -17328.76,E2 -17328.76} C_VEL
LIN {X 0,Y 277.266,Z 252.447,A -85,B 0,C 180,E1 -17332.529,E2 -17332.529} C_VEL
LIN {X 0,Y 277.303,Z 252.605,A -85,B 0,C 180,E1 -17336.406,E2 -17336.406} C_VEL
LIN {X 0,Y 279.566,Z 262.83,A -85,B 0,C 180,E1 -17340.231,E2 -17340.231} C_VEL
LIN {X 0,Y 280.507,Z 267.524,A -85,B 0,C 180,E1 -17341.821,E2 -17341.821} C_VEL
LIN {X 0,Y 282.11,Z 272.061,A -85,B 0,C 180,E1 -17342.181,E2 -17342.181} C_VEL
LIN {X 0,Y 285.73,Z 281.557,A -85,B 0,C 180,E1 -17342.778,E2 -17342.778} C_VEL
LIN {X 0,Y 290.234,Z 309.171,A -85,B 0,C 180,E1 -17343.941,E2 -17343.941} C_VEL
LIN {X 0,Y 288.317,Z 376.098,A -85,B 0,C 180,E1 -17345.662,E2 -17345.662} C_VEL
LIN {X 0,Y 287.451,Z 389.008,A -85,B 0,C 180,E1 -17346.255,E2 -17346.255} C_VEL
LIN {X 0,Y 286.285,Z 401.018,A -85,B 0,C 180,E1 -17347.062,E2 -17347.062} C_VEL
LIN {X 0,Y 284.934,Z 412.395,A -85,B 0,C 180,E1 -17348.094,E2 -17348.094} C_VEL
LIN {X 0,Y 283.255,Z 424.117,A -85,B 0,C 180,E1 -17349.483,E2 -17349.483} C_VEL
LIN {X 0,Y 281.644,Z 434.662,A -85,B 0,C 180,E1 -17351.07,E2 -17351.07} C_VEL
LIN {X 0,Y 280.154,Z 444.157,A -85,B 0,C 180,E1 -17352.856,E2 -17352.856} C_VEL
LIN {X 0,Y 278.572,Z 453.289,A -85,B 0,C 180,E1 -17355.012,E2 -17355.012} C_VEL
LIN {X 0,Y 277.24,Z 460.638,A -85,B 0,C 180,E1 -17357.183,E2 -17357.183} C_VEL
LIN {X 0,Y 276.507,Z 465.61,A -85,B 0,C 180,E1 -17359.009,E2 -17359.009} C_VEL
LIN {X 0,Y 275.841,Z 470.428,A -85,B 0,C 180,E1 -17361.206,E2 -17361.206} C_VEL
LIN {X 0,Y 275.426,Z 474.109,A -85,B 0,C 180,E1 -17363.405,E2 -17363.405} C_VEL
LIN {X 0,Y 275.231,Z 476.761,A -85,B 0,C 180,E1 -17365.605,E2 -17365.605} C_VEL
LIN {X 0,Y 275.222,Z 478.008,A -85,B 0,C 180,E1 -17367.071,E2 -17367.071} C_VEL
LIN {X 0,Y 275.231,Z 478.839,A -85,B 0,C 180,E1 -17368.536,E2 -17368.536} C_VEL
LIN {X 0,Y 275.228,Z 479.234,A -85,B 0,C 180,E1 -17369.999,E2 -17369.999} C_VEL
LIN {X 0,Y 275.231,Z 479.241,A -85,B 0,C 180,E1 -17371.462,E2 -17371.462} C_VEL
LIN {X 0,Y 275.225,Z 478.862,A -85,B 0,C 180,E1 -17372.926,E2 -17372.926} C_VEL
LIN {X 0,Y 275.329,Z 477.301,A -85,B 0,C 180,E1 -17375.402,E2 -17375.402} C_VEL
LIN {X 0,Y 275.736,Z 474.293,A -85,B 0,C 180,E1 -17378.057,E2 -17378.057} C_VEL
LIN {X 0,Y 276.351,Z 470.711,A -85,B 0,C 180,E1 -17380.253,E2 -17380.253} C_VEL
LIN {X 0,Y 277.288,Z 466.029,A -85,B 0,C 180,E1 -17382.44,E2 -17382.44} C_VEL
LIN {X 0,Y 278.872,Z 458.989,A -85,B 0,C 180,E1 -17384.969,E2 -17384.969} C_VEL
LIN {X 0,Y 280.582,Z 451.38,A -85,B 0,C 180,E1 -17387.115,E2 -17387.115} C_VEL
LIN {X 0,Y 282.51,Z 441.838,A -85,B 0,C 180,E1 -17389.244,E2 -17389.244} C_VEL
LIN {X 0,Y 284.478,Z 432.022,A -85,B 0,C 180,E1 -17390.99,E2 -17390.99} C_VEL
LIN {X 0,Y 286.615,Z 421.044,A -85,B 0,C 180,E1 -17392.527,E2 -17392.527} C_VEL
LIN {X 0,Y 288.567,Z 408.577,A -85,B 0,C 180,E1 -17393.883,E2 -17393.883} C_VEL
LIN {X 0,Y 290.201,Z 396.316,A -85,B 0,C 180,E1 -17394.883,E2 -17394.883} C_VEL
LIN {X 0,Y 291.459,Z 383.39,A -85,B 0,C 180,E1 -17395.627,E2 -17395.627} C_VEL
LIN {X 0,Y 292.386,Z 369.961,A -85,B 0,C 180,E1 -17396.107,E2 -17396.107} C_VEL
LIN {X 0,Y 294.235,Z 310.609,A -85,B 0,C 180,E1 -17397.616,E2 -17397.616} C_VEL
LIN {X 0,Y 290.653,Z 289.249,A -85,B 0,C 180,E1 -17398.665,E2 -17398.665} C_VEL
LIN {X 0,Y 285.803,Z 277.569,A -85,B 0,C 180,E1 -17399.637,E2 -17399.637} C_VEL
LIN {X 0,Y 280.832,Z 266.836,A -85,B 0,C 180,E1 -17400.693,E2 -17400.693} C_VEL
LIN {X 0,Y 278.7,Z 257.862,A -85,B 0,C 180,E1 -17404.128,E2 -17404.128} C_VEL
LIN {X 0,Y 277.298,Z 252.48,A -85,B 0,C 180,E1 -17406.473,E2 -17406.473} C_VEL
LIN {X 0,Y 277.204,Z 252.442,A -85,B 0,C 180,E1 -17410.478,E2 -17410.478} C_VEL
LIN {X 0,Y 277.198,Z 252.452,A -85,B 0,C 180,E1 -17413.198,E2 -17413.198} C_VEL
LIN {X 0,Y 277.198,Z 252.457,A -85,B 0,C 180,E1 -17417.327,E2 -17417.327} C_VEL
LIN {X 0,Y 277.254,Z 252.442,A -85,B 0,C 180,E1 -17421.793,E2 -17421.793} C_VEL
LIN {X 0,Y 277.28,Z 252.44,A -85,B 0,C 180,E1 -17424.336,E2 -17424.336} C_VEL
LIN {X 0,Y 277.242,Z 252.446,A -85,B 0,C 180,E1 -17427.832,E2 -17427.832} C_VEL
LIN {X 0,Y 277.24,Z 252.449,A -85,B 0,C 180,E1 -17431.202,E2 -17431.202} C_VEL
LIN {X 0,Y 277.246,Z 252.449,A -85,B 0,C 180,E1 -17434.468,E2 -17434.468} C_VEL
LIN {X 0,Y 277.262,Z 252.438,A -85,B 0,C 180,E1 -17437.648,E2 -17437.648} C_VEL
LIN {X 0,Y 277.328,Z 252.432,A -85,B 0,C 180,E1 -17440.76,E2 -17440.76} C_VEL
LIN {X 0,Y 277.407,Z 252.424,A -85,B 0,C 180,E1 -17445.32,E2 -17445.32} C_VEL
LIN {X 0,Y 277.453,Z 252.421,A -85,B 0,C 180,E1 -17449.782,E2 -17449.782} C_VEL
LIN {X 0,Y 277.604,Z 252.399,A -85,B 0,C 180,E1 -17452.723,E2 -17452.723} C_VEL
LIN {X 0,Y 277.801,Z 252.38,A -85,B 0,C 180,E1 -17458.545,E2 -17458.545} C_VEL
LIN {X 0,Y 277.789,Z 252.371,A -85,B 0,C 180,E1 -17461.445,E2 -17461.445} C_VEL
LIN {X 0,Y 277.587,Z 252.406,A -85,B 0,C 180,E1 -17467.267,E2 -17467.267} C_VEL
LIN {X 0,Y 277.444,Z 252.418,A -85,B 0,C 180,E1 -17470.208,E2 -17470.208} C_VEL
LIN {X 0,Y 277.4,Z 252.431,A -85,B 0,C 180,E1 -17474.67,E2 -17474.67} C_VEL
LIN {X 0,Y 277.313,Z 252.443,A -85,B 0,C 180,E1 -17479.23,E2 -17479.23} C_VEL
LIN {X 0,Y 277.266,Z 252.447,A -85,B 0,C 180,E1 -17483.92,E2 -17483.92} C_VEL
LIN {X 0,Y 277.25,Z 252.443,A -85,B 0,C 180,E1 -17487.478,E2 -17487.478} C_VEL
LIN {X 0,Y 277.226,Z 252.455,A -85,B 0,C 180,E1 -17490.468,E2 -17490.468} C_VEL
LIN {X 0,Y 277.253,Z 252.63,A -85,B 0,C 180,E1 -17492.912,E2 -17492.912} C_VEL
LIN {X 0,Y 279.406,Z 260.616,A -85,B 0,C 180,E1 -17496.15,E2 -17496.15} C_VEL
LIN {X 0,Y 283.878,Z 269.734,A -85,B 0,C 180,E1 -17497.11,E2 -17497.11} C_VEL
LIN {X 0,Y 290.514,Z 284.21,A -85,B 0,C 180,E1 -17498.411,E2 -17498.411} C_VEL
LIN {X 0,Y 293.202,Z 291.13,A -85,B 0,C 180,E1 -17498.938,E2 -17498.938} C_VEL
LIN {X 0,Y 294.606,Z 300.131,A -85,B 0,C 180,E1 -17499.365,E2 -17499.365} C_VEL
LIN {X 0,Y 292.195,Z 367.889,A -85,B 0,C 180,E1 -17501.085,E2 -17501.085} C_VEL
LIN {X 0,Y 291.182,Z 381.274,A -85,B 0,C 180,E1 -17501.681,E2 -17501.681} C_VEL
LIN {X 0,Y 289.926,Z 394.083,A -85,B 0,C 180,E1 -17502.546,E2 -17502.546} C_VEL
LIN {X 0,Y 288.411,Z 405.073,A -85,B 0,C 180,E1 -17503.538,E2 -17503.538} C_VEL
LIN {X 0,Y 286.517,Z 416.918,A -85,B 0,C 180,E1 -17504.941,E2 -17504.941} C_VEL
LIN {X 0,Y 284.519,Z 427.283,A -85,B 0,C 180,E1 -17506.487,E2 -17506.487} C_VEL
LIN {X 0,Y 282.588,Z 436.691,A -85,B 0,C 180,E1 -17508.245,E2 -17508.245} C_VEL
LIN {X 0,Y 280.665,Z 445.52,A -85,B 0,C 180,E1 -17510.32,E2 -17510.32} C_VEL
LIN {X 0,Y 279.095,Z 452.51,A -85,B 0,C 180,E1 -17512.365,E2 -17512.365} C_VEL
LIN {X 0,Y 277.818,Z 458.16,A -85,B 0,C 180,E1 -17514.422,E2 -17514.422} C_VEL
LIN {X 0,Y 276.63,Z 463.587,A -85,B 0,C 180,E1 -17516.958,E2 -17516.958} C_VEL
LIN {X 0,Y 275.917,Z 467.34,A -85,B 0,C 180,E1 -17519.376,E2 -17519.376} C_VEL
LIN {X 0,Y 275.478,Z 469.178,A -85,B 0,C 180,E1 -17521.007,E2 -17521.007} C_VEL
LIN {X 0,Y 275.039,Z 470.969,A -85,B 0,C 180,E1 -17523.409,E2 -17523.409} C_VEL
LIN {X 0,Y 274.844,Z 471.681,A -85,B 0,C 180,E1 -17525.851,E2 -17525.851} C_VEL
LIN {X 0,Y 274.83,Z 471.57,A -85,B 0,C 180,E1 -17527.446,E2 -17527.446} C_VEL
LIN {X 0,Y 274.845,Z 470.951,A -85,B 0,C 180,E1 -17529.025,E2 -17529.025} C_VEL
LIN {X 0,Y 275.072,Z 469.613,A -85,B 0,C 180,E1 -17530.947,E2 -17530.947} C_VEL
LIN {X 0,Y 275.37,Z 467.435,A -85,B 0,C 180,E1 -17532.934,E2 -17532.934} C_VEL
LIN {X 0,Y 275.924,Z 463.604,A -85,B 0,C 180,E1 -17535.413,E2 -17535.413} C_VEL
LIN {X 0,Y 276.613,Z 459.201,A -85,B 0,C 180,E1 -17537.529,E2 -17537.529} C_VEL
LIN {X 0,Y 277.541,Z 453.196,A -85,B 0,C 180,E1 -17539.791,E2 -17539.791} C_VEL
LIN {X 0,Y 278.873,Z 445.624,A -85,B 0,C 180,E1 -17542.034,E2 -17542.034} C_VEL
LIN {X 0,Y 280.187,Z 437.906,A -85,B 0,C 180,E1 -17543.882,E2 -17543.882} C_VEL
LIN {X 0,Y 281.841,Z 427.968,A -85,B 0,C 180,E1 -17545.808,E2 -17545.808} C_VEL
LIN {X 0,Y 283.422,Z 418.027,A -85,B 0,C 180,E1 -17547.336,E2 -17547.336} C_VEL
LIN {X 0,Y 285.048,Z 406.332,A -85,B 0,C 180,E1 -17548.765,E2 -17548.765} C_VEL
LIN {X 0,Y 286.439,Z 394.141,A -85,B 0,C 180,E1 -17549.913,E2 -17549.913} C_VEL
LIN {X 0,Y 287.597,Z 381.12,A -85,B 0,C 180,E1 -17550.798,E2 -17550.798} C_VEL
LIN {X 0,Y 288.475,Z 367.877,A -85,B 0,C 180,E1 -17551.397,E2 -17551.397} C_VEL
LIN {X 0,Y 290.493,Z 297.121,A -85,B 0,C 180,E1 -17553.204,E2 -17553.204} C_VEL
LIN {X 0,Y 287.674,Z 282.37,A -85,B 0,C 180,E1 -17553.861,E2 -17553.861} C_VEL
LIN {X 0,Y 282.436,Z 268.761,A -85,B 0,C 180,E1 -17554.73,E2 -17554.73} C_VEL
LIN {X 0,Y 279.237,Z 260.733,A -85,B 0,C 180,E1 -17555.316,E2 -17555.316} C_VEL
LIN {X 0,Y 277.807,Z 253.429,A -85,B 0,C 180,E1 -17557.999,E2 -17557.999} C_VEL
LIN {X 0,Y 277.563,Z 252.429,A -85,B 0,C 180,E1 -17558.556,E2 -17558.556} C_VEL
LIN {X 0,Y 277.384,Z 252.42,A -85,B 0,C 180,E1 -17563.182,E2 -17563.182} C_VEL
LIN {X 0,Y 277.37,Z 252.428,A -85,B 0,C 180,E1 -17566.185,E2 -17566.185} C_VEL
LIN {X 0,Y 277.315,Z 252.435,A -85,B 0,C 180,E1 -17570.352,E2 -17570.352} C_VEL
LIN {X 0,Y 277.249,Z 252.44,A -85,B 0,C 180,E1 -17574.154,E2 -17574.154} C_VEL
LIN {X 0,Y 277.24,Z 252.45,A -85,B 0,C 180,E1 -17577.485,E2 -17577.485} C_VEL
LIN {X 0,Y 277.212,Z 252.456,A -85,B 0,C 180,E1 -17582.169,E2 -17582.169} C_VEL
LIN {X 0,Y 277.248,Z 252.431,A -85,B 0,C 180,E1 -17585.8,E2 -17585.8} C_VEL
LIN {X 0,Y 277.193,Z 252.455,A -85,B 0,C 180,E1 -17589.336,E2 -17589.336} C_VEL
LIN {X 0,Y 277.169,Z 252.439,A -85,B 0,C 180,E1 -17593.207,E2 -17593.207} C_VEL
LIN {X 0,Y 277.173,Z 252.457,A -85,B 0,C 180,E1 -17597.336,E2 -17597.336} C_VEL
LIN {X 0,Y 277.233,Z 252.423,A -85,B 0,C 180,E1 -17601.802,E2 -17601.802} C_VEL
LIN {X 0,Y 277.262,Z 252.44,A -85,B 0,C 180,E1 -17604.346,E2 -17604.346} C_VEL
LIN {X 0,Y 277.224,Z 252.445,A -85,B 0,C 180,E1 -17607.841,E2 -17607.841} C_VEL
LIN {X 0,Y 277.205,Z 252.419,A -85,B 0,C 180,E1 -17611.21,E2 -17611.21} C_VEL
LIN {X 0,Y 277.21,Z 252.445,A -85,B 0,C 180,E1 -17614.867,E2 -17614.867} C_VEL
LIN {X 0,Y 277.275,Z 252.435,A -85,B 0,C 180,E1 -17619.222,E2 -17619.222} C_VEL
LIN {X 0,Y 277.293,Z 252.41,A -85,B 0,C 180,E1 -17621.171,E2 -17621.171} C_VEL
LIN {X 0,Y 276.608,Z 252.489,A -85,B 0,C 180,E1 -17622.384,E2 -17622.384} C_VEL
LIN {X 0,Y 273.762,Z 252.857,A -85,B 0,C 180,E1 -17624.361,E2 -17624.361} C_VEL
LIN {X 0,Y 271.39,Z 253.169,A -85,B 0,C 180,E1 -17625.968,E2 -17625.968} C_VEL
LIN {X 0,Y 270.418,Z 253.296,A -85,B 0,C 180,E1 -17627.213,E2 -17627.213} C_VEL
LIN {X 0,Y 270.361,Z 253.304,A -85,B 0,C 180,E1 -17627.634,E2 -17627.634} C_VEL
LIN {X 0,Y 270.527,Z 253.275,A -85,B 0,C 180,E1 -17631.038,E2 -17631.038} C_VEL
LIN {X 0,Y 270.509,Z 253.248,A -85,B 0,C 180,E1 -17634.04,E2 -17634.04} C_VEL
LIN {X 0,Y 270.772,Z 253.254,A -85,B 0,C 180,E1 -17638.518,E2 -17638.518} C_VEL
LIN {X 0,Y 270.776,Z 253.25,A -85,B 0,C 180,E1 -17641.492,E2 -17641.492} C_VEL
LIN {X 0,Y 270.58,Z 253.265,A -85,B 0,C 180,E1 -17647.467,E2 -17647.467} C_VEL
LIN {X 0,Y 270.417,Z 253.303,A -85,B 0,C 180,E1 -17650.487,E2 -17650.487} C_VEL
LIN {X 0,Y 270.386,Z 253.273,A -85,B 0,C 180,E1 -17655.07,E2 -17655.07} C_VEL
LIN {X 0,Y 270.271,Z 253.318,A -85,B 0,C 180,E1 -17659.762,E2 -17659.762} C_VEL
LIN {X 0,Y 270.236,Z 253.297,A -85,B 0,C 180,E1 -17664.594,E2 -17664.594} C_VEL
LIN {X 0,Y 270.211,Z 253.325,A -85,B 0,C 180,E1 -17667.92,E2 -17667.92} C_VEL
LIN {X 0,Y 270.186,Z 253.312,A -85,B 0,C 180,E1 -17671.353,E2 -17671.353} C_VEL
LIN {X 0,Y 270.21,Z 253.328,A -85,B 0,C 180,E1 -17674.909,E2 -17674.909} C_VEL
LIN {X 0,Y 270.212,Z 253.32,A -85,B 0,C 180,E1 -17678.713,E2 -17678.713} C_VEL
LIN {X 0,Y 270.162,Z 253.322,A -85,B 0,C 180,E1 -17683.247,E2 -17683.247} C_VEL
LIN {X 0,Y 270.165,Z 253.33,A -85,B 0,C 180,E1 -17687.439,E2 -17687.439} C_VEL
LIN {X 0,Y 270.207,Z 253.326,A -85,B 0,C 180,E1 -17691.373,E2 -17691.373} C_VEL
LIN {X 0,Y 270.221,Z 253.321,A -85,B 0,C 180,E1 -17695.607,E2 -17695.607} C_VEL
LIN {X 0,Y 270.299,Z 253.606,A -85,B 0,C 180,E1 -17695.957,E2 -17695.957} C_VEL
LIN {X 0,Y 272.776,Z 264.896,A -85,B 0,C 180,E1 -17700.265,E2 -17700.265} C_VEL
LIN {X 0,Y 273.302,Z 267.515,A -85,B 0,C 180,E1 -17701.126,E2 -17701.126} C_VEL
LIN {X 0,Y 275.515,Z 273.39,A -85,B 0,C 180,E1 -17701.588,E2 -17701.588} C_VEL
LIN {X 0,Y 279.574,Z 284.355,A -85,B 0,C 180,E1 -17702.294,E2 -17702.294} C_VEL
LIN {X 0,Y 283.663,Z 309.688,A -85,B 0,C 180,E1 -17703.384,E2 -17703.384} C_VEL
LIN {X 0,Y 281.828,Z 374.117,A -85,B 0,C 180,E1 -17705.064,E2 -17705.064} C_VEL
LIN {X 0,Y 280.981,Z 386.968,A -85,B 0,C 180,E1 -17705.624,E2 -17705.624} C_VEL
LIN {X 0,Y 279.687,Z 400.035,A -85,B 0,C 180,E1 -17706.489,E2 -17706.489} C_VEL
LIN {X 0,Y 278.322,Z 411.631,A -85,B 0,C 180,E1 -17707.546,E2 -17707.546} C_VEL
LIN {X 0,Y 276.6,Z 423.515,A -85,B 0,C 180,E1 -17708.967,E2 -17708.967} C_VEL
LIN {X 0,Y 274.893,Z 434.146,A -85,B 0,C 180,E1 -17710.587,E2 -17710.587} C_VEL
LIN {X 0,Y 273.332,Z 443.729,A -85,B 0,C 180,E1 -17712.414,E2 -17712.414} C_VEL
LIN {X 0,Y 271.693,Z 452.928,A -85,B 0,C 180,E1 -17714.624,E2 -17714.624} C_VEL
LIN {X 0,Y 270.297,Z 460.324,A -85,B 0,C 180,E1 -17716.848,E2 -17716.848} C_VEL
LIN {X 0,Y 269.497,Z 465.337,A -85,B 0,C 180,E1 -17718.72,E2 -17718.72} C_VEL
LIN {X 0,Y 268.789,Z 470.192,A -85,B 0,C 180,E1 -17720.973,E2 -17720.973} C_VEL
LIN {X 0,Y 268.35,Z 473.909,A -85,B 0,C 180,E1 -17723.231,E2 -17723.231} C_VEL
LIN {X 0,Y 268.146,Z 476.594,A -85,B 0,C 180,E1 -17725.489,E2 -17725.489} C_VEL
LIN {X 0,Y 268.118,Z 477.856,A -85,B 0,C 180,E1 -17726.994,E2 -17726.994} C_VEL
LIN {X 0,Y 268.137,Z 478.713,A -85,B 0,C 180,E1 -17728.497,E2 -17728.497} C_VEL
LIN {X 0,Y 268.154,Z 479.128,A -85,B 0,C 180,E1 -17729.999,E2 -17729.999} C_VEL
LIN {X 0,Y 268.137,Z 479.15,A -85,B 0,C 180,E1 -17731.501,E2 -17731.501} C_VEL
LIN {X 0,Y 268.122,Z 478.785,A -85,B 0,C 180,E1 -17733.004,E2 -17733.004} C_VEL
LIN {X 0,Y 268.22,Z 477.449,A -85,B 0,C 180,E1 -17735.288,E2 -17735.288} C_VEL
LIN {X 0,Y 268.696,Z 474.29,A -85,B 0,C 180,E1 -17738.27,E2 -17738.27} C_VEL
LIN {X 0,Y 269.341,Z 470.74,A -85,B 0,C 180,E1 -17740.523,E2 -17740.523} C_VEL
LIN {X 0,Y 270.331,Z 466.095,A -85,B 0,C 180,E1 -17742.765,E2 -17742.765} C_VEL
LIN {X 0,Y 272.023,Z 459.103,A -85,B 0,C 180,E1 -17745.355,E2 -17745.355} C_VEL
LIN {X 0,Y 273.79,Z 451.554,A -85,B 0,C 180,E1 -17747.553,E2 -17747.553} C_VEL
LIN {X 0,Y 275.432,Z 443.86,A -85,B 0,C 180,E1 -17749.371,E2 -17749.371} C_VEL
LIN {X 0,Y 277.634,Z 433.43,A -85,B 0,C 180,E1 -17751.338,E2 -17751.338} C_VEL
LIN {X 0,Y 279.864,Z 422.826,A -85,B 0,C 180,E1 -17752.906,E2 -17752.906} C_VEL
LIN {X 0,Y 281.855,Z 410.951,A -85,B 0,C 180,E1 -17754.293,E2 -17754.293} C_VEL
LIN {X 0,Y 283.69,Z 398.274,A -85,B 0,C 180,E1 -17755.396,E2 -17755.396} C_VEL
LIN {X 0,Y 285.056,Z 385.62,A -85,B 0,C 180,E1 -17756.197,E2 -17756.197} C_VEL
LIN {X 0,Y 285.996,Z 372.889,A -85,B 0,C 180,E1 -17756.715,E2 -17756.715} C_VEL
LIN {X 0,Y 288.078,Z 311.258,A -85,B 0,C 180,E1 -17758.322,E2 -17758.322} C_VEL
LIN {X 0,Y 284.734,Z 291.429,A -85,B 0,C 180,E1 -17759.345,E2 -17759.345} C_VEL
LIN {X 0,Y 279.145,Z 278.284,A -85,B 0,C 180,E1 -17760.505,E2 -17760.505} C_VEL
LIN {X 0,Y 273.671,Z 266.921,A -85,B 0,C 180,E1 -17761.705,E2 -17761.705} C_VEL
LIN {X 0,Y 272.734,Z 263.01,A -85,B 0,C 180,E1 -17763.143,E2 -17763.143} C_VEL
LIN {X 0,Y 270.267,Z 253.562,A -85,B 0,C 180,E1 -17767.197,E2 -17767.197} C_VEL
LIN {X 0,Y 270.206,Z 253.323,A -85,B 0,C 180,E1 -17768.707,E2 -17768.707} C_VEL
LIN {X 0,Y 270.155,Z 253.33,A -85,B 0,C 180,E1 -17773.241,E2 -17773.241} C_VEL
LIN {X 0,Y 270.157,Z 253.334,A -85,B 0,C 180,E1 -17777.434,E2 -17777.434} C_VEL
LIN {X 0,Y 270.197,Z 253.321,A -85,B 0,C 180,E1 -17781.368,E2 -17781.368} C_VEL
LIN {X 0,Y 270.201,Z 253.32,A -85,B 0,C 180,E1 -17785.09,E2 -17785.09} C_VEL
LIN {X 0,Y 270.187,Z 253.322,A -85,B 0,C 180,E1 -17789.132,E2 -17789.132} C_VEL
LIN {X 0,Y 270.224,Z 253.316,A -85,B 0,C 180,E1 -17792.159,E2 -17792.159} C_VEL
LIN {X 0,Y 270.228,Z 253.322,A -85,B 0,C 180,E1 -17795.538,E2 -17795.538} C_VEL
LIN {X 0,Y 270.278,Z 253.317,A -85,B 0,C 180,E1 -17800.238,E2 -17800.238} C_VEL
LIN {X 0,Y 270.375,Z 253.304,A -85,B 0,C 180,E1 -17804.929,E2 -17804.929} C_VEL
LIN {X 0,Y 270.406,Z 253.301,A -85,B 0,C 180,E1 -17809.513,E2 -17809.513} C_VEL
LIN {X 0,Y 270.565,Z 253.275,A -85,B 0,C 180,E1 -17812.533,E2 -17812.533} C_VEL
LIN {X 0,Y 270.765,Z 253.256,A -85,B 0,C 180,E1 -17818.508,E2 -17818.508} C_VEL
LIN {X 0,Y 270.753,Z 253.247,A -85,B 0,C 180,E1 -17821.482,E2 -17821.482} C_VEL
LIN {X 0,Y 270.549,Z 253.284,A -85,B 0,C 180,E1 -17827.458,E2 -17827.458} C_VEL
LIN {X 0,Y 270.397,Z 253.297,A -85,B 0,C 180,E1 -17830.477,E2 -17830.477} C_VEL
LIN {X 0,Y 270.359,Z 253.309,A -85,B 0,C 180,E1 -17835.061,E2 -17835.061} C_VEL
LIN {X 0,Y 270.247,Z 253.319,A -85,B 0,C 180,E1 -17839.754,E2 -17839.754} C_VEL
LIN {X 0,Y 270.206,Z 253.327,A -85,B 0,C 180,E1 -17844.586,E2 -17844.586} C_VEL
LIN {X 0,Y 270.178,Z 253.319,A -85,B 0,C 180,E1 -17847.912,E2 -17847.912} C_VEL
LIN {X 0,Y 270.183,Z 253.474,A -85,B 0,C 180,E1 -17851.998,E2 -17851.998} C_VEL
LIN {X 0,Y 271.97,Z 260.043,A -85,B 0,C 180,E1 -17854.864,E2 -17854.864} C_VEL
LIN {X 0,Y 272.311,Z 261.145,A -85,B 0,C 180,E1 -17855.152,E2 -17855.152} C_VEL
LIN {X 0,Y 278.332,Z 272.861,A -85,B 0,C 180,E1 -17856.453,E2 -17856.453} C_VEL
LIN {X 0,Y 284.984,Z 287.51,A -85,B 0,C 180,E1 -17857.81,E2 -17857.81} C_VEL
LIN {X 0,Y 287.35,Z 293.623,A -85,B 0,C 180,E1 -17858.299,E2 -17858.299} C_VEL
LIN {X 0,Y 288.502,Z 301.363,A -85,B 0,C 180,E1 -17858.677,E2 -17858.677} C_VEL
LIN {X 0,Y 285.98,Z 368.315,A -85,B 0,C 180,E1 -17860.411,E2 -17860.411} C_VEL
LIN {X 0,Y 284.938,Z 381.512,A -85,B 0,C 180,E1 -17861.012,E2 -17861.012} C_VEL
LIN {X 0,Y 283.657,Z 393.84,A -85,B 0,C 180,E1 -17861.857,E2 -17861.857} C_VEL
LIN {X 0,Y 282,Z 405.592,A -85,B 0,C 180,E1 -17862.941,E2 -17862.941} C_VEL
LIN {X 0,Y 280.019,Z 417.389,A -85,B 0,C 180,E1 -17864.376,E2 -17864.376} C_VEL
LIN {X 0,Y 277.932,Z 427.647,A -85,B 0,C 180,E1 -17865.944,E2 -17865.944} C_VEL
LIN {X 0,Y 276.11,Z 436.165,A -85,B 0,C 180,E1 -17867.565,E2 -17867.565} C_VEL
LIN {X 0,Y 274.081,Z 445.006,A -85,B 0,C 180,E1 -17869.651,E2 -17869.651} C_VEL
LIN {X 0,Y 272.413,Z 452.102,A -85,B 0,C 180,E1 -17871.746,E2 -17871.746} C_VEL
LIN {X 0,Y 270.783,Z 458.862,A -85,B 0,C 180,E1 -17874.271,E2 -17874.271} C_VEL
LIN {X 0,Y 269.579,Z 464,A -85,B 0,C 180,E1 -17876.808,E2 -17876.808} C_VEL
LIN {X 0,Y 268.749,Z 468.071,A -85,B 0,C 180,E1 -17879.639,E2 -17879.639} C_VEL
LIN {X 0,Y 268.191,Z 470.197,A -85,B 0,C 180,E1 -17881.857,E2 -17881.857} C_VEL
LIN {X 0,Y 267.934,Z 471.213,A -85,B 0,C 180,E1 -17883.52,E2 -17883.52} C_VEL
LIN {X 0,Y 267.78,Z 471.723,A -85,B 0,C 180,E1 -17885.172,E2 -17885.172} C_VEL
LIN {X 0,Y 267.749,Z 471.744,A -85,B 0,C 180,E1 -17886.815,E2 -17886.815} C_VEL
LIN {X 0,Y 267.717,Z 471.33,A -85,B 0,C 180,E1 -17888.439,E2 -17888.439} C_VEL
LIN {X 0,Y 267.942,Z 469.888,A -85,B 0,C 180,E1 -17890.759,E2 -17890.759} C_VEL
LIN {X 0,Y 268.347,Z 467.244,A -85,B 0,C 180,E1 -17893.258,E2 -17893.258} C_VEL
LIN {X 0,Y 268.966,Z 463.138,A -85,B 0,C 180,E1 -17895.864,E2 -17895.864} C_VEL
LIN {X 0,Y 269.661,Z 458.752,A -85,B 0,C 180,E1 -17897.967,E2 -17897.967} C_VEL
LIN {X 0,Y 270.771,Z 452.046,A -85,B 0,C 180,E1 -17900.466,E2 -17900.466} C_VEL
LIN {X 0,Y 272.097,Z 444.873,A -85,B 0,C 180,E1 -17902.581,E2 -17902.581} C_VEL
LIN {X 0,Y 273.508,Z 436.98,A -85,B 0,C 180,E1 -17904.472,E2 -17904.472} C_VEL
LIN {X 0,Y 275.15,Z 427.502,A -85,B 0,C 180,E1 -17906.309,E2 -17906.309} C_VEL
LIN {X 0,Y 276.895,Z 416.52,A -85,B 0,C 180,E1 -17908.001,E2 -17908.001} C_VEL
LIN {X 0,Y 278.652,Z 404.398,A -85,B 0,C 180,E1 -17909.459,E2 -17909.459} C_VEL
LIN {X 0,Y 280.05,Z 391.467,A -85,B 0,C 180,E1 -17910.63,E2 -17910.63} C_VEL
LIN {X 0,Y 281.178,Z 378.618,A -85,B 0,C 180,E1 -17911.467,E2 -17911.467} C_VEL
LIN {X 0,Y 281.976,Z 365.699,A -85,B 0,C 180,E1 -17912.003,E2 -17912.003} C_VEL
LIN {X 0,Y 283.981,Z 298.065,A -85,B 0,C 180,E1 -17913.752,E2 -17913.752} C_VEL
LIN {X 0,Y 281.422,Z 284.591,A -85,B 0,C 180,E1 -17914.372,E2 -17914.372} C_VEL
LIN {X 0,Y 275.668,Z 269.863,A -85,B 0,C 180,E1 -17915.35,E2 -17915.35} C_VEL
LIN {X 0,Y 272.114,Z 260.875,A -85,B 0,C 180,E1 -17916.024,E2 -17916.024} C_VEL
LIN {X 0,Y 270.917,Z 255.047,A -85,B 0,C 180,E1 -17918.197,E2 -17918.197} C_VEL
LIN {X 0,Y 270.5,Z 253.309,A -85,B 0,C 180,E1 -17919.054,E2 -17919.054} C_VEL
LIN {X 0,Y 270.326,Z 253.302,A -85,B 0,C 180,E1 -17923.533,E2 -17923.533} C_VEL
LIN {X 0,Y 270.302,Z 253.308,A -85,B 0,C 180,E1 -17926.62,E2 -17926.62} C_VEL
LIN {X 0,Y 270.242,Z 253.317,A -85,B 0,C 180,E1 -17930.592,E2 -17930.592} C_VEL
LIN {X 0,Y 270.196,Z 253.319,A -85,B 0,C 180,E1 -17934.594,E2 -17934.594} C_VEL
LIN {X 0,Y 270.167,Z 253.325,A -85,B 0,C 180,E1 -17937.922,E2 -17937.922} C_VEL
LIN {X 0,Y 270.143,Z 253.333,A -85,B 0,C 180,E1 -17941.355,E2 -17941.355} C_VEL
LIN {X 0,Y 270.173,Z 253.312,A -85,B 0,C 180,E1 -17944.911,E2 -17944.911} C_VEL
LIN {X 0,Y 270.176,Z 253.333,A -85,B 0,C 180,E1 -17948.715,E2 -17948.715} C_VEL
LIN {X 0,Y 270.126,Z 253.316,A -85,B 0,C 180,E1 -17953.25,E2 -17953.25} C_VEL
LIN {X 0,Y 270.132,Z 253.334,A -85,B 0,C 180,E1 -17957.443,E2 -17957.443} C_VEL
LIN {X 0,Y 270.176,Z 253.3,A -85,B 0,C 180,E1 -17961.377,E2 -17961.377} C_VEL
LIN {X 0,Y 270.183,Z 253.327,A -85,B 0,C 180,E1 -17965.099,E2 -17965.099} C_VEL
LIN {X 0,Y 270.159,Z 253.312,A -85,B 0,C 180,E1 -17969.147,E2 -17969.147} C_VEL
LIN {X 0,Y 270.177,Z 253.297,A -85,B 0,C 180,E1 -17972.183,E2 -17972.183} C_VEL
LIN {X 0,Y 270.175,Z 253.328,A -85,B 0,C 180,E1 -17975.569,E2 -17975.569} C_VEL
LIN {X 0,Y 270.251,Z 253.301,A -85,B 0,C 180,E1 -17980.247,E2 -17980.247} C_VEL
LIN {X 0,Y 270.365,Z 253.288,A -85,B 0,C 180,E1 -17984.939,E2 -17984.939} C_VEL
LIN {X 0,Y 270.361,Z 253.304,A -85,B 0,C 180,E1 -17987.634,E2 -17987.634} C_VEL
LIN {X 0,Y 269.786,Z 253.38,A -85,B 0,C 180,E1 -17988.878,E2 -17988.878} C_VEL
LIN {X 0,Y 267.062,Z 253.707,A -85,B 0,C 180,E1 -17990.91,E2 -17990.91} C_VEL
LIN {X 0,Y 263.817,Z 254.083,A -85,B 0,C 180,E1 -17993.406,E2 -17993.406} C_VEL
LIN {X 0,Y 263.427,Z 254.129,A -85,B 0,C 180,E1 -17994.269,E2 -17994.269} C_VEL
LIN {X 0,Y 263.736,Z 254.13,A -85,B 0,C 180,E1 -17998.478,E2 -17998.478} C_VEL
LIN {X 0,Y 263.74,Z 254.127,A -85,B 0,C 180,E1 -18001.532,E2 -18001.532} C_VEL
LIN {X 0,Y 263.542,Z 254.143,A -85,B 0,C 180,E1 -18007.667,E2 -18007.667} C_VEL
LIN {X 0,Y 263.36,Z 254.18,A -85,B 0,C 180,E1 -18010.771,E2 -18010.771} C_VEL
LIN {X 0,Y 263.333,Z 254.151,A -85,B 0,C 180,E1 -18015.484,E2 -18015.484} C_VEL
LIN {X 0,Y 263.249,Z 254.194,A -85,B 0,C 180,E1 -18020.313,E2 -18020.313} C_VEL
LIN {X 0,Y 263.179,Z 254.183,A -85,B 0,C 180,E1 -18025.299,E2 -18025.299} C_VEL
LIN {X 0,Y 263.146,Z 254.206,A -85,B 0,C 180,E1 -18028.738,E2 -18028.738} C_VEL
LIN {X 0,Y 263.141,Z 254.193,A -85,B 0,C 180,E1 -18032.292,E2 -18032.292} C_VEL
LIN {X 0,Y 263.187,Z 254.19,A -85,B 0,C 180,E1 -18036.763,E2 -18036.763} C_VEL
LIN {X 0,Y 263.105,Z 254.213,A -85,B 0,C 180,E1 -18039.878,E2 -18039.878} C_VEL
LIN {X 0,Y 263.091,Z 254.211,A -85,B 0,C 180,E1 -18043.996,E2 -18043.996} C_VEL
LIN {X 0,Y 263.095,Z 254.212,A -85,B 0,C 180,E1 -18048.419,E2 -18048.419} C_VEL
LIN {X 0,Y 263.145,Z 254.204,A -85,B 0,C 180,E1 -18052.099,E2 -18052.099} C_VEL
LIN {X 0,Y 263.219,Z 254.424,A -85,B 0,C 180,E1 -18055.374,E2 -18055.374} C_VEL
LIN {X 0,Y 265.738,Z 265.727,A -85,B 0,C 180,E1 -18059.834,E2 -18059.834} C_VEL
LIN {X 0,Y 266.124,Z 267.585,A -85,B 0,C 180,E1 -18060.401,E2 -18060.401} C_VEL
LIN {X 0,Y 273.193,Z 285.893,A -85,B 0,C 180,E1 -18061.726,E2 -18061.726} C_VEL
LIN {X 0,Y 277.234,Z 311.374,A -85,B 0,C 180,E1 -18062.85,E2 -18062.85} C_VEL
LIN {X 0,Y 275.164,Z 375.756,A -85,B 0,C 180,E1 -18064.569,E2 -18064.569} C_VEL
LIN {X 0,Y 274.2,Z 389.473,A -85,B 0,C 180,E1 -18065.233,E2 -18065.233} C_VEL
LIN {X 0,Y 272.943,Z 401.311,A -85,B 0,C 180,E1 -18066.074,E2 -18066.074} C_VEL
LIN {X 0,Y 271.501,Z 412.553,A -85,B 0,C 180,E1 -18067.151,E2 -18067.151} C_VEL
LIN {X 0,Y 269.746,Z 424.212,A -85,B 0,C 180,E1 -18068.606,E2 -18068.606} C_VEL
LIN {X 0,Y 267.982,Z 434.707,A -85,B 0,C 180,E1 -18070.265,E2 -18070.265} C_VEL
LIN {X 0,Y 266.529,Z 443.311,A -85,B 0,C 180,E1 -18071.955,E2 -18071.955} C_VEL
LIN {X 0,Y 265.027,Z 451.185,A -85,B 0,C 180,E1 -18073.832,E2 -18073.832} C_VEL
LIN {X 0,Y 263.57,Z 458.882,A -85,B 0,C 180,E1 -18076.113,E2 -18076.113} C_VEL
LIN {X 0,Y 262.499,Z 465.063,A -85,B 0,C 180,E1 -18078.415,E2 -18078.415} C_VEL
LIN {X 0,Y 261.758,Z 469.957,A -85,B 0,C 180,E1 -18080.728,E2 -18080.728} C_VEL
LIN {X 0,Y 261.277,Z 473.709,A -85,B 0,C 180,E1 -18083.046,E2 -18083.046} C_VEL
LIN {X 0,Y 261.062,Z 476.427,A -85,B 0,C 180,E1 -18085.366,E2 -18085.366} C_VEL
LIN {X 0,Y 261.018,Z 477.705,A -85,B 0,C 180,E1 -18086.912,E2 -18086.912} C_VEL
LIN {X 0,Y 261.044,Z 478.583,A -85,B 0,C 180,E1 -18088.456,E2 -18088.456} C_VEL
LIN {X 0,Y 261.082,Z 479.022,A -85,B 0,C 180,E1 -18089.999,E2 -18089.999} C_VEL
LIN {X 0,Y 261.045,Z 479.058,A -85,B 0,C 180,E1 -18091.541,E2 -18091.541} C_VEL
LIN {X 0,Y 261.08,Z 477.974,A -85,B 0,C 180,E1 -18094.631,E2 -18094.631} C_VEL
LIN {X 0,Y 261.248,Z 476.807,A -85,B 0,C 180,E1 -18096.176,E2 -18096.176} C_VEL
LIN {X 0,Y 261.643,Z 474.297,A -85,B 0,C 180,E1 -18098.494,E2 -18098.494} C_VEL
LIN {X 0,Y 262.351,Z 470.784,A -85,B 0,C 180,E1 -18100.807,E2 -18100.807} C_VEL
LIN {X 0,Y 263.391,Z 466.185,A -85,B 0,C 180,E1 -18103.108,E2 -18103.108} C_VEL
LIN {X 0,Y 265.179,Z 459.238,A -85,B 0,C 180,E1 -18105.761,E2 -18105.761} C_VEL
LIN {X 0,Y 267.011,Z 451.737,A -85,B 0,C 180,E1 -18108.014,E2 -18108.014} C_VEL
LIN {X 0,Y 268.746,Z 444.099,A -85,B 0,C 180,E1 -18109.873,E2 -18109.873} C_VEL
LIN {X 0,Y 270.841,Z 434.836,A -85,B 0,C 180,E1 -18111.7,E2 -18111.7} C_VEL
LIN {X 0,Y 273.075,Z 424.543,A -85,B 0,C 180,E1 -18113.308,E2 -18113.308} C_VEL
LIN {X 0,Y 275.151,Z 413.164,A -85,B 0,C 180,E1 -18114.723,E2 -18114.723} C_VEL
LIN {X 0,Y 277.05,Z 401.338,A -85,B 0,C 180,E1 -18115.847,E2 -18115.847} C_VEL
LIN {X 0,Y 278.607,Z 388.322,A -85,B 0,C 180,E1 -18116.75,E2 -18116.75} C_VEL
LIN {X 0,Y 279.746,Z 374.723,A -85,B 0,C 180,E1 -18117.378,E2 -18117.378} C_VEL
LIN {X 0,Y 282.04,Z 312.306,A -85,B 0,C 180,E1 -18119.047,E2 -18119.047} C_VEL
LIN {X 0,Y 278.968,Z 293.891,A -85,B 0,C 180,E1 -18120.031,E2 -18120.031} C_VEL
LIN {X 0,Y 273.496,Z 281.195,A -85,B 0,C 180,E1 -18121.208,E2 -18121.208} C_VEL
LIN {X 0,Y 268.14,Z 270.319,A -85,B 0,C 180,E1 -18122.392,E2 -18122.392} C_VEL
LIN {X 0,Y 266.355,Z 266.547,A -85,B 0,C 180,E1 -18122.882,E2 -18122.882} C_VEL
LIN {X 0,Y 264.625,Z 259.649,A -85,B 0,C 180,E1 -18125.751,E2 -18125.751} C_VEL
LIN {X 0,Y 263.186,Z 254.232,A -85,B 0,C 180,E1 -18128.335,E2 -18128.335} C_VEL
LIN {X 0,Y 263.116,Z 254.21,A -85,B 0,C 180,E1 -18131.893,E2 -18131.893} C_VEL
LIN {X 0,Y 263.085,Z 254.211,A -85,B 0,C 180,E1 -18136.157,E2 -18136.157} C_VEL
LIN {X 0,Y 263.118,Z 254.205,A -85,B 0,C 180,E1 -18140.766,E2 -18140.766} C_VEL
LIN {X 0,Y 263.16,Z 254.201,A -85,B 0,C 180,E1 -18144.013,E2 -18144.013} C_VEL
LIN {X 0,Y 263.131,Z 254.204,A -85,B 0,C 180,E1 -18147.707,E2 -18147.707} C_VEL
LIN {X 0,Y 263.149,Z 254.2,A -85,B 0,C 180,E1 -18151.801,E2 -18151.801} C_VEL
LIN {X 0,Y 263.19,Z 254.2,A -85,B 0,C 180,E1 -18155.213,E2 -18155.213} C_VEL
LIN {X 0,Y 263.243,Z 254.193,A -85,B 0,C 180,E1 -18159.687,E2 -18159.687} C_VEL
LIN {X 0,Y 263.322,Z 254.185,A -85,B 0,C 180,E1 -18164.515,E2 -18164.515} C_VEL
LIN {X 0,Y 263.345,Z 254.183,A -85,B 0,C 180,E1 -18169.228,E2 -18169.228} C_VEL
LIN {X 0,Y 263.527,Z 254.149,A -85,B 0,C 180,E1 -18172.332,E2 -18172.332} C_VEL
LIN {X 0,Y 263.728,Z 254.133,A -85,B 0,C 180,E1 -18178.468,E2 -18178.468} C_VEL
LIN {X 0,Y 263.716,Z 254.124,A -85,B 0,C 180,E1 -18181.522,E2 -18181.522} C_VEL
LIN {X 0,Y 263.513,Z 254.162,A -85,B 0,C 180,E1 -18187.658,E2 -18187.658} C_VEL
LIN {X 0,Y 263.336,Z 254.179,A -85,B 0,C 180,E1 -18190.761,E2 -18190.761} C_VEL
LIN {X 0,Y 263.3,Z 254.19,A -85,B 0,C 180,E1 -18195.475,E2 -18195.475} C_VEL
LIN {X 0,Y 263.223,Z 254.192,A -85,B 0,C 180,E1 -18200.304,E2 -18200.304} C_VEL
LIN {X 0,Y 263.149,Z 254.203,A -85,B 0,C 180,E1 -18205.291,E2 -18205.291} C_VEL
LIN {X 0,Y 263.113,Z 254.196,A -85,B 0,C 180,E1 -18208.73,E2 -18208.73} C_VEL
LIN {X 0,Y 263.143,Z 254.326,A -85,B 0,C 180,E1 -18211.012,E2 -18211.012} C_VEL
LIN {X 0,Y 264.857,Z 260.613,A -85,B 0,C 180,E1 -18213.857,E2 -18213.857} C_VEL
LIN {X 0,Y 265.76,Z 262.719,A -85,B 0,C 180,E1 -18214.204,E2 -18214.204} C_VEL
LIN {X 0,Y 271.568,Z 273.456,A -85,B 0,C 180,E1 -18215.49,E2 -18215.49} C_VEL
LIN {X 0,Y 278.056,Z 287.452,A -85,B 0,C 180,E1 -18216.883,E2 -18216.883} C_VEL
LIN {X 0,Y 281.636,Z 296.563,A -85,B 0,C 180,E1 -18217.653,E2 -18217.653} C_VEL
LIN {X 0,Y 282.455,Z 301.267,A -85,B 0,C 180,E1 -18217.906,E2 -18217.906} C_VEL
LIN {X 0,Y 279.837,Z 368.499,A -85,B 0,C 180,E1 -18219.691,E2 -18219.691} C_VEL
LIN {X 0,Y 278.754,Z 381.637,A -85,B 0,C 180,E1 -18220.302,E2 -18220.302} C_VEL
LIN {X 0,Y 277.362,Z 394.42,A -85,B 0,C 180,E1 -18221.201,E2 -18221.201} C_VEL
LIN {X 0,Y 275.611,Z 406.107,A -85,B 0,C 180,E1 -18222.314,E2 -18222.314} C_VEL
LIN {X 0,Y 273.594,Z 417.579,A -85,B 0,C 180,E1 -18223.744,E2 -18223.744} C_VEL
LIN {X 0,Y 271.385,Z 428.018,A -85,B 0,C 180,E1 -18225.378,E2 -18225.378} C_VEL
LIN {X 0,Y 269.242,Z 437.514,A -85,B 0,C 180,E1 -18227.262,E2 -18227.262} C_VEL
LIN {X 0,Y 267.104,Z 446.269,A -85,B 0,C 180,E1 -18229.442,E2 -18229.442} C_VEL
LIN {X 0,Y 265.428,Z 452.97,A -85,B 0,C 180,E1 -18231.523,E2 -18231.523} C_VEL
LIN {X 0,Y 263.747,Z 459.559,A -85,B 0,C 180,E1 -18234.112,E2 -18234.112} C_VEL
LIN {X 0,Y 262.506,Z 464.634,A -85,B 0,C 180,E1 -18236.784,E2 -18236.784} C_VEL
LIN {X 0,Y 261.741,Z 468.132,A -85,B 0,C 180,E1 -18239.327,E2 -18239.327} C_VEL
LIN {X 0,Y 261.284,Z 469.853,A -85,B 0,C 180,E1 -18241.044,E2 -18241.044} C_VEL
LIN {X 0,Y 260.954,Z 471.008,A -85,B 0,C 180,E1 -18242.754,E2 -18242.754} C_VEL
LIN {X 0,Y 260.722,Z 471.692,A -85,B 0,C 180,E1 -18244.452,E2 -18244.452} C_VEL
LIN {X 0,Y 260.64,Z 471.876,A -85,B 0,C 180,E1 -18246.443,E2 -18246.443} C_VEL
LIN {X 0,Y 260.69,Z 470.887,A -85,B 0,C 180,E1 -18249.486,E2 -18249.486} C_VEL
LIN {X 0,Y 260.897,Z 469.695,A -85,B 0,C 180,E1 -18251.142,E2 -18251.142} C_VEL
LIN {X 0,Y 261.302,Z 467.018,A -85,B 0,C 180,E1 -18253.597,E2 -18253.597} C_VEL
LIN {X 0,Y 261.908,Z 463.244,A -85,B 0,C 180,E1 -18256.026,E2 -18256.026} C_VEL
LIN {X 0,Y 262.743,Z 458.279,A -85,B 0,C 180,E1 -18258.429,E2 -18258.429} C_VEL
LIN {X 0,Y 263.834,Z 451.989,A -85,B 0,C 180,E1 -18260.804,E2 -18260.804} C_VEL
LIN {X 0,Y 265.358,Z 444.114,A -85,B 0,C 180,E1 -18263.156,E2 -18263.156} C_VEL
LIN {X 0,Y 266.845,Z 436.015,A -85,B 0,C 180,E1 -18265.091,E2 -18265.091} C_VEL
LIN {X 0,Y 268.621,Z 426.069,A -85,B 0,C 180,E1 -18267.002,E2 -18267.002} C_VEL
LIN {X 0,Y 270.486,Z 414.96,A -85,B 0,C 180,E1 -18268.699,E2 -18268.699} C_VEL
LIN {X 0,Y 272.025,Z 404.098,A -85,B 0,C 180,E1 -18270.001,E2 -18270.001} C_VEL
LIN {X 0,Y 273.481,Z 391.049,A -85,B 0,C 180,E1 -18271.198,E2 -18271.198} C_VEL
LIN {X 0,Y 274.646,Z 378.142,A -85,B 0,C 180,E1 -18272.04,E2 -18272.04} C_VEL
LIN {X 0,Y 275.48,Z 364.663,A -85,B 0,C 180,E1 -18272.591,E2 -18272.591} C_VEL
LIN {X 0,Y 277.406,Z 298.705,A -85,B 0,C 180,E1 -18274.339,E2 -18274.339} C_VEL
LIN {X 0,Y 275.071,Z 286.523,A -85,B 0,C 180,E1 -18274.918,E2 -18274.918} C_VEL
LIN {X 0,Y 268.197,Z 269.199,A -85,B 0,C 180,E1 -18276.12,E2 -18276.12} C_VEL
LIN {X 0,Y 265.079,Z 261.318,A -85,B 0,C 180,E1 -18276.734,E2 -18276.734} C_VEL
LIN {X 0,Y 264.794,Z 260.206,A -85,B 0,C 180,E1 -18276.995,E2 -18276.995} C_VEL
LIN {X 0,Y 263.484,Z 254.521,A -85,B 0,C 180,E1 -18279.324,E2 -18279.324} C_VEL
LIN {X 0,Y 263.363,Z 254.173,A -85,B 0,C 180,E1 -18279.989,E2 -18279.989} C_VEL
LIN {X 0,Y 263.273,Z 254.183,A -85,B 0,C 180,E1 -18283.903,E2 -18283.903} C_VEL
LIN {X 0,Y 263.228,Z 254.191,A -85,B 0,C 180,E1 -18287.08,E2 -18287.08} C_VEL
LIN {X 0,Y 263.171,Z 254.199,A -85,B 0,C 180,E1 -18290.844,E2 -18290.844} C_VEL
LIN {X 0,Y 263.14,Z 254.202,A -85,B 0,C 180,E1 -18295.3,E2 -18295.3} C_VEL
LIN {X 0,Y 263.096,Z 254.198,A -85,B 0,C 180,E1 -18298.741,E2 -18298.741} C_VEL
LIN {X 0,Y 263.101,Z 254.214,A -85,B 0,C 180,E1 -18302.294,E2 -18302.294} C_VEL
LIN {X 0,Y 263.132,Z 254.19,A -85,B 0,C 180,E1 -18305.988,E2 -18305.988} C_VEL
LIN {X 0,Y 263.069,Z 254.215,A -85,B 0,C 180,E1 -18309.88,E2 -18309.88} C_VEL
LIN {X 0,Y 263.056,Z 254.203,A -85,B 0,C 180,E1 -18313.999,E2 -18313.999} C_VEL
LIN {X 0,Y 263.062,Z 254.21,A -85,B 0,C 180,E1 -18318.423,E2 -18318.423} C_VEL
LIN {X 0,Y 263.114,Z 254.182,A -85,B 0,C 180,E1 -18322.103,E2 -18322.103} C_VEL
LIN {X 0,Y 263.138,Z 254.205,A -85,B 0,C 180,E1 -18325.891,E2 -18325.891} C_VEL
LIN {X 0,Y 263.097,Z 254.188,A -85,B 0,C 180,E1 -18329.507,E2 -18329.507} C_VEL
LIN {X 0,Y 263.103,Z 254.185,A -85,B 0,C 180,E1 -18333,E2 -18333} C_VEL
LIN {X 0,Y 263.11,Z 254.209,A -85,B 0,C 180,E1 -18336.387,E2 -18336.387} C_VEL
LIN {X 0,Y 263.23,Z 254.178,A -85,B 0,C 180,E1 -18339.697,E2 -18339.697} C_VEL
LIN {X 0,Y 263.307,Z 254.16,A -85,B 0,C 180,E1 -18344.525,E2 -18344.525} C_VEL
LIN {X 0,Y 263.351,Z 254.178,A -85,B 0,C 180,E1 -18349.239,E2 -18349.239} C_VEL
LIN {X 0,Y 263.525,Z 254.13,A -85,B 0,C 180,E1 -18352.343,E2 -18352.343} C_VEL
LIN {X 0,Y 263.427,Z 254.129,A -85,B 0,C 180,E1 -18354.269,E2 -18354.269} C_VEL
LIN {X 0,Y 262.689,Z 254.231,A -85,B 0,C 180,E1 -18355.548,E2 -18355.548} C_VEL
LIN {X 0,Y 259.938,Z 254.595,A -85,B 0,C 180,E1 -18357.638,E2 -18357.638} C_VEL
LIN {X 0,Y 257.683,Z 254.883,A -85,B 0,C 180,E1 -18359.336,E2 -18359.336} C_VEL
LIN {X 0,Y 256.745,Z 254.999,A -85,B 0,C 180,E1 -18360.649,E2 -18360.649} C_VEL
LIN {X 0,Y 256.68,Z 255.005,A -85,B 0,C 180,E1 -18361.093,E2 -18361.093} C_VEL
LIN {X 0,Y 256.467,Z 255.003,A -85,B 0,C 180,E1 -18366.298,E2 -18366.298} C_VEL
LIN {X 0,Y 256.435,Z 255.04,A -85,B 0,C 180,E1 -18369.47,E2 -18369.47} C_VEL
LIN {X 0,Y 256.245,Z 255.038,A -85,B 0,C 180,E1 -18374.296,E2 -18374.296} C_VEL
LIN {X 0,Y 256.187,Z 255.061,A -85,B 0,C 180,E1 -18377.569,E2 -18377.569} C_VEL
LIN {X 0,Y 256.152,Z 255.073,A -85,B 0,C 180,E1 -18381.114,E2 -18381.114} C_VEL
LIN {X 0,Y 256.145,Z 255.056,A -85,B 0,C 180,E1 -18385.115,E2 -18385.115} C_VEL
LIN {X 0,Y 256.068,Z 255.079,A -85,B 0,C 180,E1 -18389.611,E2 -18389.611} C_VEL
LIN {X 0,Y 256.08,Z 255.081,A -85,B 0,C 180,E1 -18393.296,E2 -18393.296} C_VEL
LIN {X 0,Y 256.13,Z 255.066,A -85,B 0,C 180,E1 -18397.274,E2 -18397.274} C_VEL
LIN {X 0,Y 256.032,Z 255.087,A -85,B 0,C 180,E1 -18401.213,E2 -18401.213} C_VEL
LIN {X 0,Y 256.032,Z 255.09,A -85,B 0,C 180,E1 -18405.542,E2 -18405.542} C_VEL
LIN {X 0,Y 256.033,Z 255.09,A -85,B 0,C 180,E1 -18408.791,E2 -18408.791} C_VEL
LIN {X 0,Y 256.118,Z 255.083,A -85,B 0,C 180,E1 -18412.864,E2 -18412.864} C_VEL
LIN {X 0,Y 256.151,Z 255.25,A -85,B 0,C 180,E1 -18414.757,E2 -18414.757} C_VEL
LIN {X 0,Y 258.056,Z 263.854,A -85,B 0,C 180,E1 -18418.299,E2 -18418.299} C_VEL
LIN {X 0,Y 258.86,Z 267.353,A -85,B 0,C 180,E1 -18419.585,E2 -18419.585} C_VEL
LIN {X 0,Y 263.163,Z 278.204,A -85,B 0,C 180,E1 -18420.462,E2 -18420.462} C_VEL
LIN {X 0,Y 267.049,Z 288.644,A -85,B 0,C 180,E1 -18421.19,E2 -18421.19} C_VEL
LIN {X 0,Y 270.704,Z 311.242,A -85,B 0,C 180,E1 -18422.23,E2 -18422.23} C_VEL
LIN {X 0,Y 268.673,Z 374.759,A -85,B 0,C 180,E1 -18423.961,E2 -18423.961} C_VEL
LIN {X 0,Y 267.716,Z 388.008,A -85,B 0,C 180,E1 -18424.592,E2 -18424.592} C_VEL
LIN {X 0,Y 266.308,Z 401.325,A -85,B 0,C 180,E1 -18425.542,E2 -18425.542} C_VEL
LIN {X 0,Y 264.699,Z 413.329,A -85,B 0,C 180,E1 -18426.736,E2 -18426.736} C_VEL
LIN {X 0,Y 262.899,Z 424.831,A -85,B 0,C 180,E1 -18428.227,E2 -18428.227} C_VEL
LIN {X 0,Y 261.081,Z 435.203,A -85,B 0,C 180,E1 -18429.926,E2 -18429.926} C_VEL
LIN {X 0,Y 259.361,Z 444.923,A -85,B 0,C 180,E1 -18431.944,E2 -18431.944} C_VEL
LIN {X 0,Y 257.669,Z 453.539,A -85,B 0,C 180,E1 -18434.171,E2 -18434.171} C_VEL
LIN {X 0,Y 256.217,Z 460.796,A -85,B 0,C 180,E1 -18436.516,E2 -18436.516} C_VEL
LIN {X 0,Y 255.216,Z 466.576,A -85,B 0,C 180,E1 -18438.885,E2 -18438.885} C_VEL
LIN {X 0,Y 254.52,Z 471.113,A -85,B 0,C 180,E1 -18441.263,E2 -18441.263} C_VEL
LIN {X 0,Y 254.098,Z 474.55,A -85,B 0,C 180,E1 -18443.647,E2 -18443.647} C_VEL
LIN {X 0,Y 253.989,Z 476.253,A -85,B 0,C 180,E1 -18445.237,E2 -18445.237} C_VEL
LIN {X 0,Y 253.922,Z 477.548,A -85,B 0,C 180,E1 -18446.825,E2 -18446.825} C_VEL
LIN {X 0,Y 253.954,Z 478.445,A -85,B 0,C 180,E1 -18448.413,E2 -18448.413} C_VEL
LIN {X 0,Y 253.99,Z 478.915,A -85,B 0,C 180,E1 -18449.999,E2 -18449.999} C_VEL
LIN {X 0,Y 253.955,Z 478.968,A -85,B 0,C 180,E1 -18451.584,E2 -18451.584} C_VEL
LIN {X 0,Y 253.988,Z 477.918,A -85,B 0,C 180,E1 -18454.76,E2 -18454.76} C_VEL
LIN {X 0,Y 254.179,Z 476.785,A -85,B 0,C 180,E1 -18456.348,E2 -18456.348} C_VEL
LIN {X 0,Y 254.427,Z 475.217,A -85,B 0,C 180,E1 -18457.937,E2 -18457.937} C_VEL
LIN {X 0,Y 255.078,Z 472.079,A -85,B 0,C 180,E1 -18460.315,E2 -18460.315} C_VEL
LIN {X 0,Y 256.075,Z 467.891,A -85,B 0,C 180,E1 -18462.682,E2 -18462.682} C_VEL
LIN {X 0,Y 257.414,Z 462.538,A -85,B 0,C 180,E1 -18465.031,E2 -18465.031} C_VEL
LIN {X 0,Y 259.267,Z 455.843,A -85,B 0,C 180,E1 -18467.347,E2 -18467.347} C_VEL
LIN {X 0,Y 261.294,Z 447.688,A -85,B 0,C 180,E1 -18469.611,E2 -18469.611} C_VEL
LIN {X 0,Y 263.342,Z 439.091,A -85,B 0,C 180,E1 -18471.526,E2 -18471.526} C_VEL
LIN {X 0,Y 265.778,Z 428.643,A -85,B 0,C 180,E1 -18473.367,E2 -18473.367} C_VEL
LIN {X 0,Y 268.246,Z 416.91,A -85,B 0,C 180,E1 -18474.989,E2 -18474.989} C_VEL
LIN {X 0,Y 270.263,Z 405.151,A -85,B 0,C 180,E1 -18476.235,E2 -18476.235} C_VEL
LIN {X 0,Y 271.95,Z 393,A -85,B 0,C 180,E1 -18477.198,E2 -18477.198} C_VEL
LIN {X 0,Y 273.245,Z 380.736,A -85,B 0,C 180,E1 -18477.886,E2 -18477.886} C_VEL
LIN {X 0,Y 274.099,Z 368.267,A -85,B 0,C 180,E1 -18478.321,E2 -18478.321} C_VEL
LIN {X 0,Y 276.047,Z 313.402,A -85,B 0,C 180,E1 -18479.806,E2 -18479.806} C_VEL
LIN {X 0,Y 273.247,Z 296.474,A -85,B 0,C 180,E1 -18480.742,E2 -18480.742} C_VEL
LIN {X 0,Y 267.75,Z 283.711,A -85,B 0,C 180,E1 -18481.991,E2 -18481.991} C_VEL
LIN {X 0,Y 261.004,Z 270.186,A -85,B 0,C 180,E1 -18483.565,E2 -18483.565} C_VEL
LIN {X 0,Y 259.12,Z 266.354,A -85,B 0,C 180,E1 -18484.105,E2 -18484.105} C_VEL
LIN {X 0,Y 257.067,Z 258.665,A -85,B 0,C 180,E1 -18487.542,E2 -18487.542} C_VEL
LIN {X 0,Y 256.074,Z 255.13,A -85,B 0,C 180,E1 -18489.375,E2 -18489.375} C_VEL
LIN {X 0,Y 256.035,Z 255.088,A -85,B 0,C 180,E1 -18493.33,E2 -18493.33} C_VEL
LIN {X 0,Y 256.039,Z 255.089,A -85,B 0,C 180,E1 -18497.824,E2 -18497.824} C_VEL
LIN {X 0,Y 256.07,Z 255.082,A -85,B 0,C 180,E1 -18500.852,E2 -18500.852} C_VEL
LIN {X 0,Y 256.083,Z 255.079,A -85,B 0,C 180,E1 -18504.802,E2 -18504.802} C_VEL
LIN {X 0,Y 256.086,Z 255.077,A -85,B 0,C 180,E1 -18508.566,E2 -18508.566} C_VEL
LIN {X 0,Y 256.094,Z 255.076,A -85,B 0,C 180,E1 -18512.186,E2 -18512.186} C_VEL
LIN {X 0,Y 256.134,Z 255.077,A -85,B 0,C 180,E1 -18515.691,E2 -18515.691} C_VEL
LIN {X 0,Y 256.147,Z 255.079,A -85,B 0,C 180,E1 -18519.098,E2 -18519.098} C_VEL
LIN {X 0,Y 256.257,Z 255.064,A -85,B 0,C 180,E1 -18524.077,E2 -18524.077} C_VEL
LIN {X 0,Y 256.287,Z 255.061,A -85,B 0,C 180,E1 -18528.928,E2 -18528.928} C_VEL
LIN {X 0,Y 256.468,Z 255.026,A -85,B 0,C 180,E1 -18532.12,E2 -18532.12} C_VEL
LIN {X 0,Y 256.436,Z 255.028,A -85,B 0,C 180,E1 -18536.853,E2 -18536.853} C_VEL
LIN {X 0,Y 256.69,Z 255.01,A -85,B 0,C 180,E1 -18538.426,E2 -18538.426} C_VEL
LIN {X 0,Y 256.677,Z 255,A -85,B 0,C 180,E1 -18541.564,E2 -18541.564} C_VEL
LIN {X 0,Y 256.433,Z 255.034,A -85,B 0,C 180,E1 -18546.572,E2 -18546.572} C_VEL
LIN {X 0,Y 256.415,Z 255.036,A -85,B 0,C 180,E1 -18549.46,E2 -18549.46} C_VEL
LIN {X 0,Y 256.22,Z 255.064,A -85,B 0,C 180,E1 -18554.286,E2 -18554.286} C_VEL
LIN {X 0,Y 256.165,Z 255.07,A -85,B 0,C 180,E1 -18557.559,E2 -18557.559} C_VEL
LIN {X 0,Y 256.125,Z 255.08,A -85,B 0,C 180,E1 -18561.106,E2 -18561.106} C_VEL
LIN {X 0,Y 256.114,Z 255.079,A -85,B 0,C 180,E1 -18565.107,E2 -18565.107} C_VEL
LIN {X 0,Y 256.034,Z 255.082,A -85,B 0,C 180,E1 -18569.603,E2 -18569.603} C_VEL
LIN {X 0,Y 256.079,Z 255.306,A -85,B 0,C 180,E1 -18570.05,E2 -18570.05} C_VEL
LIN {X 0,Y 257.74,Z 261.006,A -85,B 0,C 180,E1 -18572.715,E2 -18572.715} C_VEL
LIN {X 0,Y 262.16,Z 269.096,A -85,B 0,C 180,E1 -18573.837,E2 -18573.837} C_VEL
LIN {X 0,Y 268.35,Z 281.221,A -85,B 0,C 180,E1 -18575.26,E2 -18575.26} C_VEL
LIN {X 0,Y 275.114,Z 296.687,A -85,B 0,C 180,E1 -18576.771,E2 -18576.771} C_VEL
LIN {X 0,Y 276.162,Z 300.398,A -85,B 0,C 180,E1 -18577.036,E2 -18577.036} C_VEL
LIN {X 0,Y 276.462,Z 303.323,A -85,B 0,C 180,E1 -18577.171,E2 -18577.171} C_VEL
LIN {X 0,Y 273.754,Z 368.846,A -85,B 0,C 180,E1 -18578.943,E2 -18578.943} C_VEL
LIN {X 0,Y 272.52,Z 382.734,A -85,B 0,C 180,E1 -18579.61,E2 -18579.61} C_VEL
LIN {X 0,Y 271.212,Z 394.382,A -85,B 0,C 180,E1 -18580.458,E2 -18580.458} C_VEL
LIN {X 0,Y 269.262,Z 406.717,A -85,B 0,C 180,E1 -18581.659,E2 -18581.659} C_VEL
LIN {X 0,Y 267.109,Z 418.358,A -85,B 0,C 180,E1 -18583.156,E2 -18583.156} C_VEL
LIN {X 0,Y 264.867,Z 428.433,A -85,B 0,C 180,E1 -18584.785,E2 -18584.785} C_VEL
LIN {X 0,Y 262.811,Z 437.007,A -85,B 0,C 180,E1 -18586.513,E2 -18586.513} C_VEL
LIN {X 0,Y 260.743,Z 445.078,A -85,B 0,C 180,E1 -18588.519,E2 -18588.519} C_VEL
LIN {X 0,Y 258.811,Z 452.582,A -85,B 0,C 180,E1 -18590.852,E2 -18590.852} C_VEL
LIN {X 0,Y 257.268,Z 458.267,A -85,B 0,C 180,E1 -18593.061,E2 -18593.061} C_VEL
LIN {X 0,Y 255.98,Z 463.095,A -85,B 0,C 180,E1 -18595.44,E2 -18595.44} C_VEL
LIN {X 0,Y 254.873,Z 467.538,A -85,B 0,C 180,E1 -18598.407,E2 -18598.407} C_VEL
LIN {X 0,Y 254.38,Z 469.4,A -85,B 0,C 180,E1 -18600.18,E2 -18600.18} C_VEL
LIN {X 0,Y 253.913,Z 470.997,A -85,B 0,C 180,E1 -18602.325,E2 -18602.325} C_VEL
LIN {X 0,Y 253.579,Z 471.972,A -85,B 0,C 180,E1 -18605.437,E2 -18605.437} C_VEL
LIN {X 0,Y 253.545,Z 471.883,A -85,B 0,C 180,E1 -18607.167,E2 -18607.167} C_VEL
LIN {X 0,Y 253.699,Z 470.416,A -85,B 0,C 180,E1 -18610.346,E2 -18610.346} C_VEL
LIN {X 0,Y 254.103,Z 467.814,A -85,B 0,C 180,E1 -18613.119,E2 -18613.119} C_VEL
LIN {X 0,Y 254.7,Z 464.303,A -85,B 0,C 180,E1 -18615.622,E2 -18615.622} C_VEL
LIN {X 0,Y 255.485,Z 459.642,A -85,B 0,C 180,E1 -18618.095,E2 -18618.095} C_VEL
LIN {X 0,Y 256.552,Z 453.684,A -85,B 0,C 180,E1 -18620.541,E2 -18620.541} C_VEL
LIN {X 0,Y 258.063,Z 446.142,A -85,B 0,C 180,E1 -18622.962,E2 -18622.962} C_VEL
LIN {X 0,Y 259.886,Z 436.766,A -85,B 0,C 180,E1 -18625.348,E2 -18625.348} C_VEL
LIN {X 0,Y 261.694,Z 426.975,A -85,B 0,C 180,E1 -18627.308,E2 -18627.308} C_VEL
LIN {X 0,Y 263.575,Z 416.049,A -85,B 0,C 180,E1 -18629.046,E2 -18629.046} C_VEL
LIN {X 0,Y 265.213,Z 405.448,A -85,B 0,C 180,E1 -18630.381,E2 -18630.381} C_VEL
LIN {X 0,Y 266.589,Z 393.963,A -85,B 0,C 180,E1 -18631.512,E2 -18631.512} C_VEL
LIN {X 0,Y 267.88,Z 380.62,A -85,B 0,C 180,E1 -18632.465,E2 -18632.465} C_VEL
LIN {X 0,Y 268.822,Z 367.499,A -85,B 0,C 180,E1 -18633.08,E2 -18633.08} C_VEL
LIN {X 0,Y 270.941,Z 299.745,A -85,B 0,C 180,E1 -18634.927,E2 -18634.927} C_VEL
